		IF bFullPackage THEN
		//WXT530
			//Add collection WXT530
			IF GVL_Fastighet.WXT530 THEN
				M_AddJSONObject('CollectionOpen', 'WXT530');
				//Vind (aR1)
					M_AddJSONObject('DN', TO_STRING(GVL_WXT530._GW3U_DN));
					M_AddJSONObject('DM', TO_STRING(GVL_WXT530._GW3U_DM));
					M_AddJSONObject('DX', TO_STRING(GVL_WXT530._GW3U_DX));
					M_AddJSONObject('SN', TO_STRING(GVL_WXT530._GW3U_SN));
					M_AddJSONObject('SM', TO_STRING(GVL_WXT530._GW3U_SM));
					M_AddJSONObject('SX', TO_STRING(GVL_WXT530._GW3U_SX));
				//Tryck, temperatur och fuktighet (aR2)
					M_AddJSONObject('GT3U', TO_STRING(GVL_WXT530._GW3U_GT3U));
					M_AddJSONObject('GT41', TO_STRING(GVL_WXT530._GW3U_GT41));
					M_AddJSONObject('GM41', TO_STRING(GVL_WXT530._GW3U_GM41));
					M_AddJSONObject('GP41', TO_STRING(GVL_WXT530._GW3U_GP41));	
				//Nederbörd (aR3)		
					M_AddJSONObject('RC', TO_STRING(GVL_WXT530._GW3U_RC));
					M_AddJSONObject('RD', TO_STRING(GVL_WXT530._GW3U_RD));
					M_AddJSONObject('RI', TO_STRING(GVL_WXT530._GW3U_RI));
					M_AddJSONObject('HC', TO_STRING(GVL_WXT530._GW3U_HC));
					M_AddJSONObject('HD', TO_STRING(GVL_WXT530._GW3U_HD));
					M_AddJSONObject('HI', TO_STRING(GVL_WXT530._GW3U_HI));
					M_AddJSONObject('RP', TO_STRING(GVL_WXT530._GW3U_RP));
					M_AddJSONObject('HP', TO_STRING(GVL_WXT530._GW3U_HP));		
			//Close collection WXT530
				M_AddJSONObject('CollectionClose',',');
			END_IF
		//IO
			//Add collection IO
				M_AddJSONObject('CollectionOpen', 'IO');
				// Analog in, hårdvara
					//M_AddJSONObject('AI1', TO_STRING(GVL_IO._AI1));
					//M_AddJSONObject('AI2', TO_STRING(GVL_IO._AI2));
					//M_AddJSONObject('AI3', TO_STRING(GVL_IO._AI3));
					//M_AddJSONObject('AI4', TO_STRING(GVL_IO._AI4));
					//M_AddJSONObject('AI5', TO_STRING(GVL_IO._AI5));
					//M_AddJSONObject('AI6', TO_STRING(GVL_IO._AI6));
					//M_AddJSONObject('AI7', TO_STRING(GVL_IO._AI7));
					//M_AddJSONObject('AI8', TO_STRING(GVL_IO._AI8));
				// Analog in
					M_AddJSONObject('GT41_MV', TO_STRING(GVL_IO._GT41_MV / 100)); //Scaled to degrees celsius, PT1000 temp sensor at F15
					M_AddJSONObject('GT42_MV', TO_STRING(GVL_IO._GT42_MV / 100)); //Scaled to degrees celsius, PT1000 temp sensor at F15
					M_AddJSONObject('GT43_MV', TO_STRING(GVL_IO._GT43_MV));
					M_AddJSONObject('GT44_MV', TO_STRING(GVL_IO._GT44_MV));
					M_AddJSONObject('GT45_MV', TO_STRING(GVL_IO._GT45_MV));
					M_AddJSONObject('GT46_MV', TO_STRING(GVL_IO._GT46_MV));
					M_AddJSONObject('GT47_MV', TO_STRING(GVL_IO._GT47_MV));
					M_AddJSONObject('GT48_MV', TO_STRING(GVL_IO._GT48_MV));
			//Close collection IO
				M_AddJSONObject('CollectionClose',',');				
		END_IF
		//ClusterControl
			//Add new collection ClusterControl
				M_AddJSONObject('CollectionOpen', 'ClusterControl');		
				//V1
					//M_AddJSONObject('V1_IT', TO_STRING(GVL_ClusterCtrl._CCtrl_V1_IT));
					M_AddJSONObject('V1_P', TO_STRING(GVL_ClusterCtrl._CCtrl_V1_P));
					M_AddJSONObject('V1_P1', TO_STRING(GVL_ClusterCtrl._CCtrl_V1_P1));
					M_AddJSONObject('V1_P2', TO_STRING(GVL_ClusterCtrl._CCtrl_V1_P2));
					M_AddJSONObject('V1_P3', TO_STRING(GVL_ClusterCtrl._CCtrl_V1_P3));
					M_AddJSONObject('V1_U1_L1_N', TO_STRING(GVL_ClusterCtrl._CCtrl_V1_U1_L1_N));
					M_AddJSONObject('V1_U2_L2_N', TO_STRING(GVL_ClusterCtrl._CCtrl_V1_U2_L2_N));
					M_AddJSONObject('V1_U3_L3_N', TO_STRING(GVL_ClusterCtrl._CCtrl_V1_U3_L3_N));
					M_AddJSONObject('V1_U1_L1_L2', TO_STRING(GVL_ClusterCtrl._CCtrl_V1_U1_L1_L2));
					M_AddJSONObject('V1_U2_L2_L3', TO_STRING(GVL_ClusterCtrl._CCtrl_V1_U2_L2_L3));
					M_AddJSONObject('V1_U3_L3_L1', TO_STRING(GVL_ClusterCtrl._CCtrl_V1_U3_L3_L1));
					M_AddJSONObject('V1_Itot', TO_STRING(GVL_ClusterCtrl._CCtrl_V1_Itot));
					M_AddJSONObject('V1_I1', TO_STRING(GVL_ClusterCtrl._CCtrl_V1_I1));
					M_AddJSONObject('V1_I2', TO_STRING(GVL_ClusterCtrl._CCtrl_V1_I2));
					M_AddJSONObject('V1_I3', TO_STRING(GVL_ClusterCtrl._CCtrl_V1_I3));
					//M_AddJSONObject('V1_Yield_Wh', TO_STRING(GVL_ClusterCtrl._CCtrl_V1_Yield_Wh));
					M_AddJSONObject('V1_Yield_kWh', TO_STRING(GVL_ClusterCtrl._CCtrl_V1_Yield_kWh));
					M_AddJSONObject('V1_Yield_MWh', TO_STRING(GVL_ClusterCtrl._CCtrl_V1_Yield_MWh));
					//M_AddJSONObject('V1_YieldDay_Wh', TO_STRING(GVL_ClusterCtrl._CCtrl_V1_YieldDay_Wh));
					M_AddJSONObject('V1_YieldDay_kWh', TO_STRING(GVL_ClusterCtrl._CCtrl_V1_YieldDay_kWh));
					M_AddJSONObject('V1_PV', TO_STRING(GVL_ClusterCtrl._CCtrl_V1_PV));	
					M_AddJSONObject('V1_HZ', TO_STRING(GVL_ClusterCtrl._CCtrl_V1_HZ));			
				//V2
					//M_AddJSONObject('V2_IT', TO_STRING(GVL_ClusterCtrl._CCtrl_V2_IT));
					M_AddJSONObject('V2_P', TO_STRING(GVL_ClusterCtrl._CCtrl_V2_P));
					M_AddJSONObject('V2_P1', TO_STRING(GVL_ClusterCtrl._CCtrl_V2_P1));
					M_AddJSONObject('V2_P2', TO_STRING(GVL_ClusterCtrl._CCtrl_V2_P2));
					M_AddJSONObject('V2_P3', TO_STRING(GVL_ClusterCtrl._CCtrl_V2_P3));
					M_AddJSONObject('V2_U1_L1_N', TO_STRING(GVL_ClusterCtrl._CCtrl_V2_U1_L1_N));
					M_AddJSONObject('V2_U2_L2_N', TO_STRING(GVL_ClusterCtrl._CCtrl_V2_U2_L2_N));
					M_AddJSONObject('V2_U3_L3_N', TO_STRING(GVL_ClusterCtrl._CCtrl_V2_U3_L3_N));
					M_AddJSONObject('V2_U1_L1_L2', TO_STRING(GVL_ClusterCtrl._CCtrl_V2_U1_L1_L2));
					M_AddJSONObject('V2_U2_L2_L3', TO_STRING(GVL_ClusterCtrl._CCtrl_V2_U2_L2_L3));
					M_AddJSONObject('V2_U3_L3_L1', TO_STRING(GVL_ClusterCtrl._CCtrl_V2_U3_L3_L1));
					M_AddJSONObject('V2_Itot', TO_STRING(GVL_ClusterCtrl._CCtrl_V2_Itot));
					M_AddJSONObject('V2_I1', TO_STRING(GVL_ClusterCtrl._CCtrl_V2_I1));
					M_AddJSONObject('V2_I2', TO_STRING(GVL_ClusterCtrl._CCtrl_V2_I2));
					M_AddJSONObject('V2_I3', TO_STRING(GVL_ClusterCtrl._CCtrl_V2_I3));
					//M_AddJSONObject('V2_Yield_Wh', TO_STRING(GVL_ClusterCtrl._CCtrl_V2_Yield_Wh));
					M_AddJSONObject('V2_Yield_kWh', TO_STRING(GVL_ClusterCtrl._CCtrl_V2_Yield_kWh));
					M_AddJSONObject('V2_Yield_MWh', TO_STRING(GVL_ClusterCtrl._CCtrl_V2_Yield_MWh));
					//M_AddJSONObject('V2_YieldDay_Wh', TO_STRING(GVL_ClusterCtrl._CCtrl_V2_YieldDay_Wh));
					M_AddJSONObject('V2_YieldDay_kWh', TO_STRING(GVL_ClusterCtrl._CCtrl_V2_YieldDay_kWh));
					M_AddJSONObject('V2_PV', TO_STRING(GVL_ClusterCtrl._CCtrl_V2_PV));	
					M_AddJSONObject('V2_HZ', TO_STRING(GVL_ClusterCtrl._CCtrl_V2_HZ));	
				//V3
					//M_AddJSONObject('V3_IT', TO_STRING(GVL_ClusterCtrl._CCtrl_V3_IT));
					M_AddJSONObject('V3_P', TO_STRING(GVL_ClusterCtrl._CCtrl_V3_P));
					M_AddJSONObject('V3_P1', TO_STRING(GVL_ClusterCtrl._CCtrl_V3_P1));
					M_AddJSONObject('V3_P2', TO_STRING(GVL_ClusterCtrl._CCtrl_V3_P2));
					M_AddJSONObject('V3_P3', TO_STRING(GVL_ClusterCtrl._CCtrl_V3_P3));
					M_AddJSONObject('V3_U1_L1_N', TO_STRING(GVL_ClusterCtrl._CCtrl_V3_U1_L1_N));
					M_AddJSONObject('V3_U2_L2_N', TO_STRING(GVL_ClusterCtrl._CCtrl_V3_U2_L2_N));
					M_AddJSONObject('V3_U3_L3_N', TO_STRING(GVL_ClusterCtrl._CCtrl_V3_U3_L3_N));
					M_AddJSONObject('V3_U1_L1_L2', TO_STRING(GVL_ClusterCtrl._CCtrl_V3_U1_L1_L2));
					M_AddJSONObject('V3_U2_L2_L3', TO_STRING(GVL_ClusterCtrl._CCtrl_V3_U2_L2_L3));
					M_AddJSONObject('V3_U3_L3_L1', TO_STRING(GVL_ClusterCtrl._CCtrl_V3_U3_L3_L1));
					M_AddJSONObject('V3_Itot', TO_STRING(GVL_ClusterCtrl._CCtrl_V3_Itot));
					M_AddJSONObject('V3_I1', TO_STRING(GVL_ClusterCtrl._CCtrl_V3_I1));
					M_AddJSONObject('V3_I2', TO_STRING(GVL_ClusterCtrl._CCtrl_V3_I2));
					M_AddJSONObject('V3_I3', TO_STRING(GVL_ClusterCtrl._CCtrl_V3_I3));
					//M_AddJSONObject('V3_Yield_Wh', TO_STRING(GVL_ClusterCtrl._CCtrl_V3_Yield_Wh));
					M_AddJSONObject('V3_Yield_kWh', TO_STRING(GVL_ClusterCtrl._CCtrl_V3_Yield_kWh));
					M_AddJSONObject('V3_Yield_MWh', TO_STRING(GVL_ClusterCtrl._CCtrl_V3_Yield_MWh));
					//M_AddJSONObject('V3_YieldDay_Wh', TO_STRING(GVL_ClusterCtrl._CCtrl_V3_YieldDay_Wh));
					M_AddJSONObject('V3_YieldDay_kWh', TO_STRING(GVL_ClusterCtrl._CCtrl_V3_YieldDay_kWh));
					M_AddJSONObject('V3_PV', TO_STRING(GVL_ClusterCtrl._CCtrl_V3_PV));	
					M_AddJSONObject('V3_HZ', TO_STRING(GVL_ClusterCtrl._CCtrl_V3_HZ));	
			//Close collection ClusterControl
				M_AddJSONObject('CollectionClose',',');	
		//MX41
			//Add new collection MX41
				M_AddJSONObject('CollectionOpen', 'MX41');
				//MX41 Data
					M_AddJSONObject('I1', TO_STRING(GVL_MX41._I1));
					M_AddJSONObject('I2', TO_STRING(GVL_MX41._I2));
					M_AddJSONObject('I3', TO_STRING(GVL_MX41._I3));
					M_AddJSONObject('U1_U2', TO_STRING(GVL_MX41._U1_U2));
					M_AddJSONObject('U2_U3', TO_STRING(GVL_MX41._U2_U3));
					M_AddJSONObject('U3_U1', TO_STRING(GVL_MX41._U3_U1));
					M_AddJSONObject('U1_N', TO_STRING(GVL_MX41._U1_N));
					M_AddJSONObject('U2_N', TO_STRING(GVL_MX41._U2_N));
					M_AddJSONObject('U3_N', TO_STRING(GVL_MX41._U3_N));
					M_AddJSONObject('P1', TO_STRING(GVL_MX41._P1));
					M_AddJSONObject('P2', TO_STRING(GVL_MX41._P2));
					M_AddJSONObject('P3', TO_STRING(GVL_MX41._P3));
					M_AddJSONObject('P', TO_STRING(GVL_MX41._P));
					M_AddJSONObject('PVAR', TO_STRING(GVL_MX41._PVAR));
					M_AddJSONObject('PVA', TO_STRING(GVL_MX41._PVA));
					M_AddJSONObject('PFA', TO_STRING(GVL_MX41._Pfa));
					M_AddJSONObject('HZ', TO_STRING(GVL_MX41._HZ));
					M_AddJSONObject('WHAI', TO_STRING(GVL_MX41._WHAI));
					M_AddJSONObject('WHAE', TO_STRING(GVL_MX41._WHAE));
					M_AddJSONObject('VARHI', TO_STRING(GVL_MX41._VARHI));
					M_AddJSONObject('VARHE', TO_STRING(GVL_MX41._VARHE));
					M_AddJSONObject('WHPAI', TO_STRING(GVL_MX41._WHPAI));
					M_AddJSONObject('WHPAE', TO_STRING(GVL_MX41._WHPAE));
					M_AddJSONObject('WHAEI1', TO_STRING(GVL_MX41._WHAEI1));
					M_AddJSONObject('WHAEI2', TO_STRING(GVL_MX41._WHAEI2));
					M_AddJSONObject('WHAEI3', TO_STRING(GVL_MX41._WHAEI3));
			//Close collection MX41	
				M_AddJSONObject('CollectionClose',',');	
		//SR05 Hukseflux Solar Irradiance meter
		IF GVL_Fastighet.SMAIrrMeter THEN
			//Add collection SR05
				M_AddJSONObject('CollectionOpen', 'SR05');
				//SR05 Sensor Outputs
					M_AddJSONObject('Irr', TO_STRING(GVL_SR05._SolarIrr));
					M_AddJSONObject('BT', TO_STRING(GVL_SR05._BodyTemp));
					M_AddJSONObject('ER', TO_STRING(GVL_SR05._ElecResistance));
					M_AddJSONObject('VO', TO_STRING(GVL_SR05._VoltageOutput));					
			//Close collection SR05
				M_AddJSONObject('End', sCurlyBracketEnd);
		END_IF
	//Close collection DataList	
		M_AddJSONObject('End', sCurlyBracketEnd);	
	//////////////////////////////////////////
	
	//End Collection
	M_AddJSONObject('End', sCurlyBracketEnd);	

	//Done
	M_BuildPayload := TRUE;
END_METHOD

METHOD M_ConnectMQTT : BOOL
VAR_INPUT
END_VAR
bConnect := TRUE;
END_METHOD

METHOD M_CreatePayload : BOOL
VAR_INPUT
	bFullPackage : BOOL;
END_VAR
VAR
	nLastPosAdded : DINT;
	i : DINT;
	sStringCheck : STRING;
	M_Payload_SMAClusterCntrl: INT;
END_VAR
// Method for building the Payload message that is going to be sent to the Azure IoT Hub. 
// Maximum 4kB message 
		
//Clear Payload before creating a new one
uPayload := GVL_IoT.uPayloadEmpty;

//Start Collection
M_AddJSONObject('Start', sCurlyBracket);

//General
M_AddJSONObject('ID', GVL_Fastighet.FastighetsBeteckning);
M_AddJSONObject('timeStamp', sJSONTime);

//Add new collection DataList
M_AddJSONObject('CollectionOpen', 'DataList');

(* Add the units payload that are enabled *)
IF bFullPackage THEN
	
	IF GVL_Fastighet.WXT530 THEN
		M_Payload_WXT530();
	END_IF
	
	IF GVL_Fastighet.IO THEN
		M_Payload_IO();
	END_IF
	
END_IF

IF GVL_Fastighet.SMAClusterCntrl THEN
		M_Payload_SMACluster();
END_IF

IF GVL_Fastighet.EnergyMeter THEN
	M_Payload_MX41_iEM3255();
END_IF

IF GVL_Fastighet.SR05 THEN
	M_Payload_SR05();
END_IF

//Trim the payload char ',' from last unit added to create a valid json
//Check first empty position in the array
FOR i:=0 TO SIZEOF(uPayLoad.aPayload) / SIZEOF(uPayload.aPayload[0]) DO
	IF uPayload.aPayload[i] = 0 THEN
		nLastPosAdded := i;
		EXIT;
	END_IF
END_FOR

//Remove the last ',' char to make a valid json-string
uPayload.aPayload[nLastPosAdded - 1] := 0;


//Close collection DataList	
M_AddJSONObject('End', sCurlyBracketEnd);	

//End Collection
M_AddJSONObject('End', sCurlyBracketEnd);	

//Done
M_CreatePayload := TRUE;
END_METHOD

METHOD M_Deque : BOOL
VAR
	i : INT;
END_VAR
FOR i:=0 TO GVL_IoT.nMaxPayloadBuffer DO

	//If there is data, publish it! 
	IF MEMCMP(ADR(GVL_IoT.uPayloadQueue[i]), ADR(GVL_IoT.uPayloadEmpty), SIZEOF(GVL_IoT.uPayloadEmpty)) <> 0 THEN
		//Call Publish 
		M_Publish(GVL_IoT.uPayloadQueue[i]);
		//After the publish; remove it from the queue
		GVL_IoT.uPayloadQueue[i] := GVL_IoT.uPayloadEmpty;
	END_IF

END_FOR

//Done
M_Deque := TRUE;
END_METHOD

METHOD M_DisconnectMQTT : BOOL
VAR_INPUT
END_VAR
bConnect := FALSE;
END_METHOD

METHOD M_Initialize : BOOL
VAR_INPUT
END_VAR
//Initialize startup parameters

	//Message topic that is used for every message, should not be changed! Only if the deviceName have changed
	sTopicPub := GVL_Fastighet.IoTTopicPub;
	
	//Set the SAS token
	fbMqttClient.sHostName := GVL_Fastighet.IoTHostName;
	fbMqttClient.nHostPort := GVL_Fastighet.IoTHostPort;
	//fbMqttClient.stTLS.sAzureSas := 'HostName=StunsSolarHub.azure-devices.net;DeviceId=SE_UPP_A001P001;SharedAccessSignature=SharedAccessSignature sr=StunsSolarHub.azure-devices.net%2Fdevices%2FSE_UPP_A001P001&sig=PNxS244bUszDXJ%2BMNceHTcws%2BEW3ixqGkw0V7mblAEw%3D&se=1525956832';
	//fbMqttClient.stTLS.sCA := 'c:\TwinCAT\3.1\Config\Certificates\azure.crt';
	
	//Default Publish time
	tPublishTime(PT:=GVL_Fastighet.PublishTime);

	//Set Active flag
	bActive:= TRUE;

//Initialize completed
	bInitDone := TRUE;
END_METHOD

METHOD M_Payload_IO : BOOL
VAR_INPUT
END_VAR
//IO
//Add collection IO
M_AddJSONObject('CollectionOpen', 'IO');
// Analog in
M_AddJSONObject('GT41_MV', TO_STRING(GVL_IO._GT41_MV / 100)); //Scaled to degrees celsius, PT1000 temp sensor at F15
M_AddJSONObject('GT42_MV', TO_STRING(GVL_IO._GT42_MV / 100)); //Scaled to degrees celsius, PT1000 temp sensor at F15
M_AddJSONObject('GT43_MV', TO_STRING(GVL_IO._GT43_MV));
M_AddJSONObject('GT44_MV', TO_STRING(GVL_IO._GT44_MV));
M_AddJSONObject('GT45_MV', TO_STRING(GVL_IO._GT45_MV));
M_AddJSONObject('GT46_MV', TO_STRING(GVL_IO._GT46_MV));
M_AddJSONObject('GT47_MV', TO_STRING(GVL_IO._GT47_MV));
M_AddJSONObject('GT48_MV', TO_STRING(GVL_IO._GT48_MV));
//Close collection IO
M_AddJSONObject('CollectionClose',',');
END_METHOD

METHOD M_Payload_MX41_iEM3255 : BOOL
VAR_INPUT
END_VAR
//Add collection MX41
M_AddJSONObject('CollectionOpen', 'MX41');

//MX41 Data - Schneider
M_AddJSONObject('I1', TO_STRING(GVL_MX41._I1));
M_AddJSONObject('I2', TO_STRING(GVL_MX41._I2));
M_AddJSONObject('I3', TO_STRING(GVL_MX41._I3));
M_AddJSONObject('U1_U2', TO_STRING(GVL_MX41._U1_U2));
M_AddJSONObject('U2_U3', TO_STRING(GVL_MX41._U2_U3));
M_AddJSONObject('U3_U1', TO_STRING(GVL_MX41._U3_U1));
(*The following voltage values only returns 0 at F15 per 20017-09-01, investigate and remove commentation when working. Possibly lack of N leader to meter!*)
//M_AddJSONObject('U1_N', TO_STRING(GVL_MX41._U1_N));
//M_AddJSONObject('U2_N', TO_STRING(GVL_MX41._U2_N));
//M_AddJSONObject('U3_N', TO_STRING(GVL_MX41._U3_N));
(*The following power values only returns 0 at F15 per 20017-09-01, investigate and remove commentation when working. Possibly lack of N leader to meter!*)
//M_AddJSONObject('P1', TO_STRING(GVL_MX41._P1));
//M_AddJSONObject('P2', TO_STRING(GVL_MX41._P2));
//M_AddJSONObject('P3', TO_STRING(GVL_MX41._P3));
M_AddJSONObject('P', TO_STRING(GVL_MX41._P));
M_AddJSONObject('PVAR', TO_STRING(GVL_MX41._PVAR));
M_AddJSONObject('PVA', TO_STRING(GVL_MX41._PVA));
M_AddJSONObject('PFA', TO_STRING(GVL_MX41._Pfa));
M_AddJSONObject('HZ', TO_STRING(GVL_MX41._HZ));
M_AddJSONObject('WHAI', TO_STRING(GVL_MX41._WHAI));
M_AddJSONObject('WHAE', TO_STRING(GVL_MX41._WHAE));
M_AddJSONObject('VARHI', TO_STRING(GVL_MX41._VARHI));
M_AddJSONObject('VARHE', TO_STRING(GVL_MX41._VARHE));
M_AddJSONObject('WHPAI', TO_STRING(GVL_MX41._WHPAI));
M_AddJSONObject('WHPAE', TO_STRING(GVL_MX41._WHPAE));
M_AddJSONObject('WHAEI1', TO_STRING(GVL_MX41._WHAEI1));
M_AddJSONObject('WHAEI2', TO_STRING(GVL_MX41._WHAEI2));
M_AddJSONObject('WHAEI3', TO_STRING(GVL_MX41._WHAEI3));

//Close collection MX41	
M_AddJSONObject('CollectionClose',',');
END_METHOD

METHOD M_Payload_SMACluster : BOOL
VAR_INPUT
END_VAR
//Add new collection ClusterControl
M_AddJSONObject('CollectionOpen', 'ClusterControl');		


//V1 - Inverter 1
//M_AddJSONObject('V1_IT', TO_STRING(GVL_ClusterCtrl._CCtrl_V1_IT));
M_AddJSONObject('V1_P', TO_STRING(GVL_ClusterCtrl._CCtrl_V1_P));
M_AddJSONObject('V1_P1', TO_STRING(GVL_ClusterCtrl._CCtrl_V1_P1));
M_AddJSONObject('V1_P2', TO_STRING(GVL_ClusterCtrl._CCtrl_V1_P2));
M_AddJSONObject('V1_P3', TO_STRING(GVL_ClusterCtrl._CCtrl_V1_P3));
M_AddJSONObject('V1_U1_L1_N', TO_STRING(GVL_ClusterCtrl._CCtrl_V1_U1_L1_N));
M_AddJSONObject('V1_U2_L2_N', TO_STRING(GVL_ClusterCtrl._CCtrl_V1_U2_L2_N));
M_AddJSONObject('V1_U3_L3_N', TO_STRING(GVL_ClusterCtrl._CCtrl_V1_U3_L3_N));
(*The following voltage values only returns false values at F15 per 20017-09-01, investigate and remove commentation when working*)
//M_AddJSONObject('V1_U1_L1_L2', TO_STRING(GVL_ClusterCtrl._CCtrl_V1_U1_L1_L2));
//M_AddJSONObject('V1_U2_L2_L3', TO_STRING(GVL_ClusterCtrl._CCtrl_V1_U2_L2_L3));
//M_AddJSONObject('V1_U3_L3_L1', TO_STRING(GVL_ClusterCtrl._CCtrl_V1_U3_L3_L1));
(*The following parameter Itot only returns a false value at F15 per 20017-09-01, investigate and remove commentation when working*)
//M_AddJSONObject('V1_Itot', TO_STRING(GVL_ClusterCtrl._CCtrl_V1_Itot));
M_AddJSONObject('V1_I1', TO_STRING(GVL_ClusterCtrl._CCtrl_V1_I1));
M_AddJSONObject('V1_I2', TO_STRING(GVL_ClusterCtrl._CCtrl_V1_I2));
M_AddJSONObject('V1_I3', TO_STRING(GVL_ClusterCtrl._CCtrl_V1_I3));
//M_AddJSONObject('V1_Yield_Wh', TO_STRING(GVL_ClusterCtrl._CCtrl_V1_Yield_Wh));
M_AddJSONObject('V1_Yield_kWh', TO_STRING(GVL_ClusterCtrl._CCtrl_V1_Yield_kWh));
M_AddJSONObject('V1_Yield_MWh', TO_STRING(GVL_ClusterCtrl._CCtrl_V1_Yield_MWh));
//M_AddJSONObject('V1_YieldDay_Wh', TO_STRING(GVL_ClusterCtrl._CCtrl_V1_YieldDay_Wh));
M_AddJSONObject('V1_YieldDay_kWh', TO_STRING(GVL_ClusterCtrl._CCtrl_V1_YieldDay_kWh));
(*The following parameter PV only returns a false value at F15 per 20017-09-01, investigate and remove commentation when working*)
//M_AddJSONObject('V1_PV', TO_STRING(GVL_ClusterCtrl._CCtrl_V1_PV));	
M_AddJSONObject('V1_HZ', TO_STRING(GVL_ClusterCtrl._CCtrl_V1_HZ));			


//V2 - Inverter 2
//M_AddJSONObject('V2_IT', TO_STRING(GVL_ClusterCtrl._CCtrl_V2_IT));
M_AddJSONObject('V2_P', TO_STRING(GVL_ClusterCtrl._CCtrl_V2_P));
M_AddJSONObject('V2_P1', TO_STRING(GVL_ClusterCtrl._CCtrl_V2_P1));
M_AddJSONObject('V2_P2', TO_STRING(GVL_ClusterCtrl._CCtrl_V2_P2));
M_AddJSONObject('V2_P3', TO_STRING(GVL_ClusterCtrl._CCtrl_V2_P3));
M_AddJSONObject('V2_U1_L1_N', TO_STRING(GVL_ClusterCtrl._CCtrl_V2_U1_L1_N));
M_AddJSONObject('V2_U2_L2_N', TO_STRING(GVL_ClusterCtrl._CCtrl_V2_U2_L2_N));
M_AddJSONObject('V2_U3_L3_N', TO_STRING(GVL_ClusterCtrl._CCtrl_V2_U3_L3_N));
(*The following voltage values only return false values at F15 per 20017-09-01, investigate and remove commentation when working*)
//M_AddJSONObject('V2_U1_L1_L2', TO_STRING(GVL_ClusterCtrl._CCtrl_V2_U1_L1_L2));
//M_AddJSONObject('V2_U2_L2_L3', TO_STRING(GVL_ClusterCtrl._CCtrl_V2_U2_L2_L3));
//M_AddJSONObject('V2_U3_L3_L1', TO_STRING(GVL_ClusterCtrl._CCtrl_V2_U3_L3_L1));
(*The following parameter Itot only returns a false value at F15 per 20017-09-01, investigate and remove commentation when working*)
//M_AddJSONObject('V2_Itot', TO_STRING(GVL_ClusterCtrl._CCtrl_V2_Itot));
M_AddJSONObject('V2_I1', TO_STRING(GVL_ClusterCtrl._CCtrl_V2_I1));
M_AddJSONObject('V2_I2', TO_STRING(GVL_ClusterCtrl._CCtrl_V2_I2));
M_AddJSONObject('V2_I3', TO_STRING(GVL_ClusterCtrl._CCtrl_V2_I3));
//M_AddJSONObject('V2_Yield_Wh', TO_STRING(GVL_ClusterCtrl._CCtrl_V2_Yield_Wh));
M_AddJSONObject('V2_Yield_kWh', TO_STRING(GVL_ClusterCtrl._CCtrl_V2_Yield_kWh));
M_AddJSONObject('V2_Yield_MWh', TO_STRING(GVL_ClusterCtrl._CCtrl_V2_Yield_MWh));
//M_AddJSONObject('V2_YieldDay_Wh', TO_STRING(GVL_ClusterCtrl._CCtrl_V2_YieldDay_Wh));
M_AddJSONObject('V2_YieldDay_kWh', TO_STRING(GVL_ClusterCtrl._CCtrl_V2_YieldDay_kWh));
(*The following parameter PV only returns a false value at F15 per 20017-09-01, investigate and remove commentation when working*)
//M_AddJSONObject('V2_PV', TO_STRING(GVL_ClusterCtrl._CCtrl_V2_PV));	
M_AddJSONObject('V2_HZ', TO_STRING(GVL_ClusterCtrl._CCtrl_V2_HZ));	

//V3 - Inverter 3
//M_AddJSONObject('V3_IT', TO_STRING(GVL_ClusterCtrl._CCtrl_V3_IT));
M_AddJSONObject('V3_P', TO_STRING(GVL_ClusterCtrl._CCtrl_V3_P));
M_AddJSONObject('V3_P1', TO_STRING(GVL_ClusterCtrl._CCtrl_V3_P1));
M_AddJSONObject('V3_P2', TO_STRING(GVL_ClusterCtrl._CCtrl_V3_P2));
M_AddJSONObject('V3_P3', TO_STRING(GVL_ClusterCtrl._CCtrl_V3_P3));
M_AddJSONObject('V3_U1_L1_N', TO_STRING(GVL_ClusterCtrl._CCtrl_V3_U1_L1_N));
M_AddJSONObject('V3_U2_L2_N', TO_STRING(GVL_ClusterCtrl._CCtrl_V3_U2_L2_N));
M_AddJSONObject('V3_U3_L3_N', TO_STRING(GVL_ClusterCtrl._CCtrl_V3_U3_L3_N));
(*The following voltage values only return false values at F15 per 20017-09-01, investigate and remove commentation when working*)
//M_AddJSONObject('V3_U1_L1_L2', TO_STRING(GVL_ClusterCtrl._CCtrl_V3_U1_L1_L2));
//M_AddJSONObject('V3_U2_L2_L3', TO_STRING(GVL_ClusterCtrl._CCtrl_V3_U2_L2_L3));
//M_AddJSONObject('V3_U3_L3_L1', TO_STRING(GVL_ClusterCtrl._CCtrl_V3_U3_L3_L1));
(*The following parameter Itot only returns a false value at F15 per 20017-09-01, investigate and remove commentation when working*)
//M_AddJSONObject('V3_Itot', TO_STRING(GVL_ClusterCtrl._CCtrl_V3_Itot));
M_AddJSONObject('V3_I1', TO_STRING(GVL_ClusterCtrl._CCtrl_V3_I1));
M_AddJSONObject('V3_I2', TO_STRING(GVL_ClusterCtrl._CCtrl_V3_I2));
M_AddJSONObject('V3_I3', TO_STRING(GVL_ClusterCtrl._CCtrl_V3_I3));
//M_AddJSONObject('V3_Yield_Wh', TO_STRING(GVL_ClusterCtrl._CCtrl_V3_Yield_Wh));
M_AddJSONObject('V3_Yield_kWh', TO_STRING(GVL_ClusterCtrl._CCtrl_V3_Yield_kWh));
M_AddJSONObject('V3_Yield_MWh', TO_STRING(GVL_ClusterCtrl._CCtrl_V3_Yield_MWh));
//M_AddJSONObject('V3_YieldDay_Wh', TO_STRING(GVL_ClusterCtrl._CCtrl_V3_YieldDay_Wh));
M_AddJSONObject('V3_YieldDay_kWh', TO_STRING(GVL_ClusterCtrl._CCtrl_V3_YieldDay_kWh));
(*The following parameter PV only returns a false value at F15 per 20017-09-01, investigate and remove commentation when working*)
//M_AddJSONObject('V3_PV', TO_STRING(GVL_ClusterCtrl._CCtrl_V3_PV));	
M_AddJSONObject('V3_HZ', TO_STRING(GVL_ClusterCtrl._CCtrl_V3_HZ));	


//Close collection ClusterControl
M_AddJSONObject('CollectionClose',',');
END_METHOD

METHOD M_Payload_SMAIrrMeter : BOOL
VAR_INPUT
END_VAR
END_METHOD

METHOD M_Payload_SR05 : BOOL
VAR_INPUT
END_VAR
//SR05 Hukseflux Solar Irradiance meter
//Add collection SR05
M_AddJSONObject('CollectionOpen', 'SR05');
//SR05 Sensor Outputs
M_AddJSONObject('Irr', TO_STRING(GVL_SR05._SolarIrr));
M_AddJSONObject('TempBody', TO_STRING(GVL_SR05._BodyTemp));
M_AddJSONObject('ElectricalRes', TO_STRING(GVL_SR05._ElecResistance));
M_AddJSONObject('VoltageOutput', TO_STRING(GVL_SR05._VoltageOutput));					
//Close collection SR05
M_AddJSONObject('CollectionClose',',');
END_METHOD

METHOD M_Payload_WXT530 : BOOL
VAR_INPUT
END_VAR
//WXT530
//Add collection WXT530
M_AddJSONObject('CollectionOpen', 'WXT530');
//Vind (aR1)
M_AddJSONObject('DN', TO_STRING(GVL_WXT530._GW3U_DN));
M_AddJSONObject('DM', TO_STRING(GVL_WXT530._GW3U_DM));
M_AddJSONObject('DX', TO_STRING(GVL_WXT530._GW3U_DX));
M_AddJSONObject('SN', TO_STRING(GVL_WXT530._GW3U_SN));
M_AddJSONObject('SM', TO_STRING(GVL_WXT530._GW3U_SM));
M_AddJSONObject('SX', TO_STRING(GVL_WXT530._GW3U_SX));
//Tryck, temperatur och fuktighet (aR2)
M_AddJSONObject('GT3U', TO_STRING(GVL_WXT530._GW3U_GT3U));
M_AddJSONObject('GT41', TO_STRING(GVL_WXT530._GW3U_GT41));
M_AddJSONObject('GM41', TO_STRING(GVL_WXT530._GW3U_GM41));
M_AddJSONObject('GP41', TO_STRING(GVL_WXT530._GW3U_GP41));	
//Nederbörd (aR3)		
M_AddJSONObject('RC', TO_STRING(GVL_WXT530._GW3U_RC));
M_AddJSONObject('RD', TO_STRING(GVL_WXT530._GW3U_RD));
M_AddJSONObject('RI', TO_STRING(GVL_WXT530._GW3U_RI));
M_AddJSONObject('HC', TO_STRING(GVL_WXT530._GW3U_HC));
M_AddJSONObject('HD', TO_STRING(GVL_WXT530._GW3U_HD));
M_AddJSONObject('HI', TO_STRING(GVL_WXT530._GW3U_HI));
M_AddJSONObject('RP', TO_STRING(GVL_WXT530._GW3U_RP));
M_AddJSONObject('HP', TO_STRING(GVL_WXT530._GW3U_HP));		
//Close collection WXT530
M_AddJSONObject('CollectionClose',',');
END_METHOD

METHOD M_Publish : BOOL
VAR_INPUT
	uPayloadToPublish : U_Payload;
END_VAR
//Publish the payload
fbMqttClient.Publish(sTopic:= sTopicPub, 
									pPayload:= ADR(uPayloadToPublish.aPayload), 
									nPayloadSize:= SIZEOF(uPayloadToPublish.aPayload), 
									eQoS:= TcIotMqttQos.AtMostOnceDelivery, 
									bRetain:= FALSE, 
									bQueue:= FALSE );
//Update last published time
sLastPublishedTime := sSystemTime;		
//Increase the Publish counter
GVL_IoT.nTotalMessagePublished := GVL_IoT.nTotalMessagePublished + 1;
//Done								
M_Publish := TRUE;
END_METHOD

METHOD M_Queue : BOOL
VAR_INPUT
	uPayloadQueue : U_Payload;
END_VAR
//Check where to add it
IF GVL_IoT.nLastPos < GVL_IoT.nMaxPayloadBuffer THEN
	GVL_IoT.uPayloadQueue[GVL_IoT.nLastPos] := uPayloadQueue; //Add to buffer
END_IF

IF (GVL_IoT.nLastPos + 1) = GVL_IoT.nMaxPayloadBuffer THEN
	GVL_IoT.bBufferFull := TRUE;
ELSE
	GVL_IoT.bBufferFull := FALSE;
END_IF

//Done
M_Queue := TRUE;
END_METHOD

METHOD M_QueueBufferStatus
VAR
	i : INT;
END_VAR
//Check first empty position in the array
FOR i:=0 TO GVL_IoT.nMaxPayloadBuffer DO
	IF MEMCMP(ADR(GVL_IoT.uPayloadQueue[i]), ADR(GVL_IoT.uPayloadEmpty), SIZEOF(GVL_IoT.uPayloadEmpty)) = 1 THEN
		GVL_IoT.nLastPos := i;
		EXIT;
	END_IF
END_FOR

IF MEMCMP(ADR(GVL_IoT.uPayloadQueue[0]), ADR(GVL_IoT.uPayloadEmpty), SIZEOF(GVL_IoT.uPayloadEmpty)) = 1 THEN
	GVL_IoT.bBufferEmpty := TRUE;
ELSE
	GVL_IoT.bBufferEmpty := FALSE;
END_IF
END_METHOD

END_FUNCTION_BLOCK

// ---- POUs/Loggning/iEM3255_Logg.TcPOU
PROGRAM iEM3255_Logg
VAR
	
	fbLogg1 		:FB_SaveToCSV_Schneider;
	tUpdateTime1	:TIME:=T#5S;
	sFileName1		:STRING(255):='Schneider1';
	
	fbLogg2 		:FB_SaveToCSV_Schneider;
	tUpdateTime2	:TIME:=T#5S;
	sFileName2		:STRING(255):='Schneider2';
	
	fbLogg3 		:FB_SaveToCSV_Schneider;
	tUpdateTime3	:TIME:=T#5S;
	sFileName3		:STRING(255):='Schneider3';
	
	fbLogg4 		:FB_SaveToCSV_Schneider;
	tUpdateTime4	:TIME:=T#5S;
	sFileName4		:STRING(255):='Schneider4';

	
END_VAR

fbLogg1(
	bChangeSeparatorToComma:= FALSE, 
	bExecute:= GVL_Fastighet.CSVEnergyMeter, 
	tUpdateTime:= tUpdateTime1, 
	sFileName:= sFileName1, 
	nDayOfWeek:= PLC_TID.fbTime.systemTime.wDayOfWeek,
	sColumn1TimeStamp:= PLC_TID.systemTime, 
	sColumn2:= REAL_TO_STRING(GVL_MX41._I1), 
	sColumn3:= REAL_TO_STRING(GVL_MX41._I2), 
	sColumn4:= REAL_TO_STRING(GVL_MX41._I3), 
	sColumn5:= REAL_TO_STRING(GVL_MX41._U1_U2), 
	sColumn6:= REAL_TO_STRING(GVL_MX41._U2_U3), 
	sColumn7:= REAL_TO_STRING(GVL_MX41._U3_U1));
	
fbLogg2(
	bChangeSeparatorToComma:= FALSE, 
	bExecute:= GVL_Fastighet.CSVEnergyMeter, 
	tUpdateTime:= tUpdateTime2, 
	sFileName:= sFileName2, 
	nDayOfWeek:= PLC_TID.fbTime.systemTime.wDayOfWeek,
	sColumn1TimeStamp:= PLC_TID.systemTime, 
	sColumn2:= REAL_TO_STRING(GVL_MX41._P1), 
	sColumn3:= REAL_TO_STRING(GVL_MX41._P2), 
	sColumn4:= REAL_TO_STRING(GVL_MX41._P3), 
	sColumn5:= REAL_TO_STRING(GVL_MX41._PVAR), 
	sColumn6:= REAL_TO_STRING(GVL_MX41._PVA), 
	sColumn7:= REAL_TO_STRING(GVL_MX41._Pfa));
	
fbLogg3(
	bChangeSeparatorToComma:= FALSE, 
	bExecute:= GVL_Fastighet.CSVEnergyMeter, 
	tUpdateTime:= tUpdateTime3, 
	sFileName:= sFileName3, 
	nDayOfWeek:= PLC_TID.fbTime.systemTime.wDayOfWeek,
	sColumn1TimeStamp:= PLC_TID.systemTime, 
	sColumn2:= REAL_TO_STRING(GVL_MX41._HZ), 
	sColumn3:= REAL_TO_STRING(GVL_MX41._WHAI), 
	sColumn4:= REAL_TO_STRING(GVL_MX41._WHAE), 
	sColumn5:= REAL_TO_STRING(GVL_MX41._VARHI), 
	sColumn6:= REAL_TO_STRING(GVL_MX41._VARHE), 
	sColumn7:= REAL_TO_STRING(GVL_MX41._WHPAI));
	
fbLogg4(
	bChangeSeparatorToComma:= FALSE, 
	bExecute:= GVL_Fastighet.CSVEnergyMeter, 
	tUpdateTime:= tUpdateTime4, 
	sFileName:= sFileName4, 
	nDayOfWeek:= PLC_TID.fbTime.systemTime.wDayOfWeek,
	sColumn1TimeStamp:= PLC_TID.systemTime, 
	sColumn2:= REAL_TO_STRING(GVL_MX41._WHPAE), 
	sColumn3:= REAL_TO_STRING(GVL_MX41._WHAEI1), 
	sColumn4:= REAL_TO_STRING(GVL_MX41._WHAEI2), 
	sColumn5:= REAL_TO_STRING(GVL_MX41._WHAEI3),
	sColumn6:= REAL_TO_STRING(GVL_MX41._P));

END_PROGRAM

// ---- POUs/_FBs/FB_SaveToCSV_Schneider.TcPOU
FUNCTION_BLOCK FB_SaveToCSV_Schneider
VAR CONSTANT
	MAX_CSV_COLUMNS 	: UDINT := 7;
END_VAR
VAR_INPUT
	(*	In USA/UK the CSV field separator is a comma.
	In Germany and some other European countries the CSV field separator is a semicolon. *)
	bChangeSeparatorToComma	: BOOL := FALSE;
	bExecute : BOOL;
	tUpdateTime : TIME:=T#1S; //Update time 
	sFileName	: T_MaxString := 'DefaultName';(* CSV destination file path and name *)
	nDayOfWeek : WORD;
	sColumn1TimeStamp : T_MaxString;
	sColumn2 : STRING;
	sColumn3 : STRING;
	sColumn4 : STRING; 
	sColumn5 : STRING;
	sColumn6 : STRING;
	sColumn7 : STRING;
END_VAR
VAR
	sNetId			: T_AmsNetId := '';	(* TwinCAT system network address *)	
	sCSVLine		: T_MaxString := '';(* Single CSV text line (row, record), we are using string as record buffer (your are able to see created fields) *)
	sCSVField		: T_MaxString := '';(* Single CSV field value (column, record field) *)
	bBusy			: BOOL;
	bError			: BOOL;
	nErrId			: UDINT;
	nColumn		: UDINT 	:= 1;(* Column number (record field) *)
	hFile			: UINT		:= 0;(* File handle of the source file *)
	step			: DWORD 	:= 0;
	fbFileOpen	: FB_FileOpen;(* Opens file *)
	fbFileClose	: FB_FileClose;(* Closes file *)
	fbFilePuts		: FB_FilePuts;(* Writes one record (line) *)
	fbWriter		: FB_CSVMemBufferWriter;(* Helper function block used to create CSV data bytes (single record line) *)	
	tUpdateTimer : TON;
	sCompleteFileName : STRING;
	sPathName : T_MaxString;
	sTempDate : STRING;
	sDate : STRING;
	bWeekUpdate : BOOL;
END_VAR

(* Call the timer every plc-cycle *)
tUpdateTimer(IN:=NOT tUpdateTimer.Q, PT:=tUpdateTime);


(* Update filename *)
IF nDayOfWeek = 1 AND bWeekUpdate THEN //1=Monday	
		sCompleteFileName	:= sFileName;
		sTempDate := DELETE(sColumn1TimeStamp, 16,11); //Cut the timestamp so we only save the date
		sDate := INSERT(sTempDate, '_', 10); //Add '-' after the date for seperation
		sPathName:=CONCAT(CONCAT('C:\Loggning\Schneider\',CONCAT(sDate,sFileName)),'.csv');
		bWeekUpdate := FALSE;
ELSE
	(* Update if name has changed *)
	IF sCompleteFileName <> sFileName THEN
		sCompleteFileName := sFileName;
		sTempDate := DELETE(sColumn1TimeStamp, 16,11); //Cut the timestamp so we only save the date
		sDate := INSERT(sTempDate, '_', 10); //Add '-' after the date for seperation
		sPathName:=CONCAT(CONCAT('C:\Loggning\Schneider\',CONCAT(sDate,sCompleteFileName)),'.csv');
	END_IF	
END_IF

IF nDayOfWeek <> 1 THEN
	bWeekUpdate := TRUE;
END_IF

CASE step OF
	0:	(* Wait for rising edge at bWrite variable *)
		IF bExecute AND tUpdateTimer.Q THEN
			bBusy 		:= TRUE;
			bError		:= FALSE;
			nErrId		:= 0;
			hFile			:= 0;
			step 		:= 1;
		END_IF

	1:	(* Open source file *)
		fbFileOpen(  bExecute := FALSE  );
		fbFileOpen( 	sNetId := sNetId, sPathName := sPathName, nMode := FOPEN_MODEAPPEND OR FOPEN_MODETEXT,(* Open file in TEXT mode! *)
						ePath := PATH_GENERIC, bExecute := TRUE );
		step := 2;

	2:(* Wait until open not busy *)
		fbFileOpen( bExecute := FALSE, bError => bError, nErrID => nErrID, hFile => hFile );
		IF NOT fbFileOpen.bBusy THEN
			IF NOT fbFileOpen.bError THEN
				step := 3;
			ELSE(* Error: file not found? *)
				step := 100;
			END_IF
		END_IF
		
	3:(* Convert one PLC record to CSV format *)
		sCSVLine := '';
		fbWriter.eCmd := eEnumCmd_First;(* Write first field value *)
		
		FOR nColumn := 1 TO MAX_CSV_COLUMNS BY 1 DO
				
				IF nColumn = 1 THEN
					sCSVField := STRING_TO_CSVFIELD(sColumn1TimeStamp, FALSE);
				ELSIF nColumn = 2 THEN
					sCSVField := STRING_TO_CSVFIELD(sColumn2, FALSE);
				ELSIF nColumn = 3 THEN
					sCSVField := STRING_TO_CSVFIELD(sColumn3, FALSE);
				ELSIF nColumn = 4 THEN
					sCSVField := STRING_TO_CSVFIELD(sColumn4, FALSE);
				ELSIF nColumn = 5 THEN
					sCSVField := STRING_TO_CSVFIELD(sColumn5, FALSE);
				ELSIF nColumn = 6 THEN	
					sCSVField := STRING_TO_CSVFIELD(sColumn6, FALSE);
				ELSIF nColumn = 7 THEN	
					sCSVField := STRING_TO_CSVFIELD(sColumn7, FALSE);
				END_IF
				
				(* Add new field to the record buffer *)
				fbWriter( 	pBuffer := ADR( sCSVLine ), cbBuffer := SIZEOF( sCSVLine ) - 1, putValue := sCSVField, pValue := 0, cbValue := 0,
							bCRLF := ( nColumn = MAX_CSV_COLUMNS ) );
										
				IF fbWriter.bOk THEN
					fbWriter.eCmd := eEnumCmd_Next;(* Write next field value *)
				ELSE(* Error *)
					step := 100;
					RETURN;
				END_IF

		END_FOR

		(* FB_FilePuts adds allready CR (carriage return) to the written line.
		We have to replace the $R$L characters with $L character to avoid double CR. *)
		IF RIGHT( sCSVLine, 2 ) = '$R$L' THEN
			sCSVLine := REPLACE( sCSVLine, '$L', 2, LEN( sCSVLine ) - 1 );
		END_IF

		step := 4;(* Write record to the file *)
		
	4:	(* Write single text line *)
		fbFilePuts( bExecute := FALSE );
		fbFilePuts( sNetId := sNetId, hFile := hFile, sLine := sCSVLine, bExecute := TRUE );
		step := 5;

	5:(* Wait until write not busy *)
		fbFilePuts( bExecute := FALSE, bError => bError, nErrID => nErrID );
		IF NOT fbFilePuts.bBusy THEN
			IF NOT fbFilePuts.bError THEN
				step := 10;(* Close file *)
			ELSE(* Error *)
				step := 100;
			END_IF
		END_IF

	10:	(* Close source file *)
		fbFileClose( bExecute := FALSE );
		fbFileClose( sNetId := sNetId, hFile := hFile, bExecute := TRUE );
		step := 11;

	11:(* Wait until close not busy *)
		fbFileClose( bExecute := FALSE, bError => bError, nErrID => nErrID );
		IF ( NOT fbFileClose.bBusy ) THEN
			hFile := 0;
			step := 100;
		END_IF

	100: (* Error or ready step => cleanup *)
		IF ( hFile <> 0 ) THEN
			step := 10; (* Close the source file *)
		ELSE
			bBusy := FALSE;
			step := 0;	(* Ready *)
		END_IF

END_CASE

END_FUNCTION_BLOCK

// ---- POUs/Loggning/Cluster_Logg.TcPOU
PROGRAM Cluster_Logg
VAR
	
fbLogg1 		:FB_SaveToCSV_ClusterCtrl;
	tUpdateTime1	:TIME:=T#5S;
	sFileName1		:STRING(255):='Unit1_1';
	
	fbLogg2 		:FB_SaveToCSV_ClusterCtrl;
	tUpdateTime2	:TIME:=T#5S;
	sFileName2		:STRING(255):='Unit1_2';
	
	fbLogg3 		:FB_SaveToCSV_ClusterCtrl;
	tUpdateTime3	:TIME:=T#5S;
	sFileName3		:STRING(255):='Unit1_3';
	
END_VAR

fbLogg1(
	bChangeSeparatorToComma:= FALSE, 
	bExecute:= GVL_Fastighet.CSVClusterCtrl, 
	tUpdateTime:= tUpdateTime1, 
	sFileName:= sFileName1, 
	nDayOfWeek:= PLC_TID.fbTime.systemTime.wDayOfWeek,
	sColumn1TimeStamp:= PLC_TID.systemTime, 
	sColumn2:= REAL_TO_STRING(GVL_ClusterCtrl._CCtrl_V1_P1), 
	sColumn3:= REAL_TO_STRING(GVL_ClusterCtrl._CCtrl_V1_P2), 
	sColumn4:= REAL_TO_STRING(GVL_ClusterCtrl._CCtrl_V1_P3), 
	sColumn5:= REAL_TO_STRING(GVL_ClusterCtrl._CCtrl_V1_U1_L1_N), 
	sColumn6:= REAL_TO_STRING(GVL_ClusterCtrl._CCtrl_V1_U2_L2_N), 
	sColumn7:= REAL_TO_STRING(GVL_ClusterCtrl._CCtrl_V1_U3_L3_N),
	sColumn8:= REAL_TO_STRING(GVL_ClusterCtrl._CCtrl_V1_HZ));
	
	fbLogg2(
	bChangeSeparatorToComma:= FALSE, 
	bExecute:= GVL_Fastighet.CSVClusterCtrl, 
	tUpdateTime:= tUpdateTime2, 
	sFileName:= sFileName2, 
	nDayOfWeek:= PLC_TID.fbTime.systemTime.wDayOfWeek,
	sColumn1TimeStamp:= PLC_TID.systemTime, 
	sColumn2:= REAL_TO_STRING(GVL_ClusterCtrl._CCtrl_V1_U1_L1_L2), 
	sColumn3:= REAL_TO_STRING(GVL_ClusterCtrl._CCtrl_V1_U2_L2_L3), 
	sColumn4:= REAL_TO_STRING(GVL_ClusterCtrl._CCtrl_V1_U3_L3_L1), 
	sColumn5:= REAL_TO_STRING(GVL_ClusterCtrl._CCtrl_V1_Itot),
	sColumn6:= REAL_TO_STRING(GVL_ClusterCtrl._CCtrl_V1_I1), 
	sColumn7:= REAL_TO_STRING(GVL_ClusterCtrl._CCtrl_V1_I2), 
	sColumn8:= REAL_TO_STRING(GVL_ClusterCtrl._CCtrl_V1_I3));
	
	fbLogg3(
	bChangeSeparatorToComma:= FALSE, 
	bExecute:= GVL_Fastighet.CSVClusterCtrl, 
	tUpdateTime:= tUpdateTime3, 
	sFileName:= sFileName3, 
	nDayOfWeek:= PLC_TID.fbTime.systemTime.wDayOfWeek,
	sColumn1TimeStamp:= PLC_TID.systemTime, 
	sColumn2:= REAL_TO_STRING(GVL_ClusterCtrl._CCtrl_V1_Yield_Wh), 
	sColumn3:= REAL_TO_STRING(GVL_ClusterCtrl._CCtrl_V1_Yield_kWh), 
	sColumn4:= REAL_TO_STRING(GVL_ClusterCtrl._CCtrl_V1_Yield_MWh), 
	sColumn5:= REAL_TO_STRING(GVL_ClusterCtrl._CCtrl_V1_YieldDay_Wh), 
	sColumn6:= REAL_TO_STRING(GVL_ClusterCtrl._CCtrl_V1_YieldDay_kWh), 
	sColumn7:= REAL_TO_STRING(GVL_ClusterCtrl._CCtrl_V1_P));

END_PROGRAM

// ---- POUs/_FBs/FB_SaveToCSV_ClusterCtrl.TcPOU
FUNCTION_BLOCK FB_SaveToCSV_ClusterCtrl
VAR CONSTANT
	MAX_CSV_COLUMNS 	: UDINT := 8;
END_VAR
VAR_INPUT
	(*	In USA/UK the CSV field separator is a comma.
	In Germany and some other European countries the CSV field separator is a semicolon. *)
	bChangeSeparatorToComma	: BOOL := FALSE;
	bExecute : BOOL;
	tUpdateTime : TIME:=T#1S; //Update time 
	sFileName	: T_MaxString := 'DefaultName';(* CSV destination file path and name *)
	nDayOfWeek : WORD;
	sColumn1TimeStamp : T_MaxString;
	sColumn2 : STRING;
	sColumn3 : STRING;
	sColumn4 : STRING; 
	sColumn5 : STRING;
	sColumn6 : STRING;
	sColumn7 : STRING;
	sColumn8 : STRING;
END_VAR
VAR
	sNetId			: T_AmsNetId := '';	(* TwinCAT system network address *)	
	sCSVLine		: T_MaxString := '';(* Single CSV text line (row, record), we are using string as record buffer (your are able to see created fields) *)
	sCSVField		: T_MaxString := '';(* Single CSV field value (column, record field) *)
	bBusy			: BOOL;
	bError			: BOOL;
	nErrId			: UDINT;
	nColumn		: UDINT 	:= 1;(* Column number (record field) *)
	hFile			: UINT		:= 0;(* File handle of the source file *)
	step			: DWORD 	:= 0;
	fbFileOpen	: FB_FileOpen;(* Opens file *)
	fbFileClose	: FB_FileClose;(* Closes file *)
	fbFilePuts		: FB_FilePuts;(* Writes one record (line) *)
	fbWriter		: FB_CSVMemBufferWriter;(* Helper function block used to create CSV data bytes (single record line) *)	
	tUpdateTimer : TON;
	sCompleteFileName : STRING;
	sPathName : T_MaxString;
	sTempDate : STRING;
	sDate : STRING;
	bWeekUpdate : BOOL;
END_VAR

(* Call the timer every plc-cycle *)
tUpdateTimer(IN:=NOT tUpdateTimer.Q, PT:=tUpdateTime);


(* Update filename *)
IF nDayOfWeek = 1 AND bWeekUpdate THEN //1=Monday	
		sCompleteFileName	:= sFileName;
		sTempDate := DELETE(sColumn1TimeStamp, 16,11); //Cut the timestamp so we only save the date
		sDate := INSERT(sTempDate, '_', 10); //Add '-' after the date for seperation
		sPathName:=CONCAT(CONCAT('C:\Loggning\Cluster\',CONCAT(sDate,sFileName)),'.csv');
		bWeekUpdate := FALSE;
ELSE
	(* Update if name has changed *)
	IF sCompleteFileName <> sFileName THEN
		sCompleteFileName := sFileName;
		sTempDate := DELETE(sColumn1TimeStamp, 16,11); //Cut the timestamp so we only save the date
		sDate := INSERT(sTempDate, '_', 10); //Add '-' after the date for seperation
		sPathName:=CONCAT(CONCAT('C:\Loggning\Cluster\',CONCAT(sDate,sCompleteFileName)),'.csv');
	END_IF	
END_IF

IF nDayOfWeek <> 1 THEN
	bWeekUpdate := TRUE;
END_IF

CASE step OF
	0:	(* Wait for rising edge at bWrite variable *)
		IF bExecute AND tUpdateTimer.Q THEN
			bBusy 		:= TRUE;
			bError		:= FALSE;
			nErrId		:= 0;
			hFile			:= 0;
			step 		:= 1;
		END_IF

	1:	(* Open source file *)
		fbFileOpen(  bExecute := FALSE  );
		fbFileOpen( 	sNetId := sNetId, sPathName := sPathName, nMode := FOPEN_MODEAPPEND OR FOPEN_MODETEXT,(* Open file in TEXT mode! *)
						ePath := PATH_GENERIC, bExecute := TRUE );
		step := 2;

	2:(* Wait until open not busy *)
		fbFileOpen( bExecute := FALSE, bError => bError, nErrID => nErrID, hFile => hFile );
		IF NOT fbFileOpen.bBusy THEN
			IF NOT fbFileOpen.bError THEN
				step := 3;
			ELSE(* Error: file not found? *)
				step := 100;
			END_IF
		END_IF
		
	3:(* Convert one PLC record to CSV format *)
		sCSVLine := '';
		fbWriter.eCmd := eEnumCmd_First;(* Write first field value *)
		
		FOR nColumn := 1 TO MAX_CSV_COLUMNS BY 1 DO
				
				IF nColumn = 1 THEN
					sCSVField := STRING_TO_CSVFIELD(sColumn1TimeStamp, FALSE);
				ELSIF nColumn = 2 THEN
					sCSVField := STRING_TO_CSVFIELD(sColumn2, FALSE);
				ELSIF nColumn = 3 THEN
					sCSVField := STRING_TO_CSVFIELD(sColumn3, FALSE);
				ELSIF nColumn = 4 THEN
					sCSVField := STRING_TO_CSVFIELD(sColumn4, FALSE);
				ELSIF nColumn = 5 THEN
					sCSVField := STRING_TO_CSVFIELD(sColumn5, FALSE);
				ELSIF nColumn = 6 THEN	
					sCSVField := STRING_TO_CSVFIELD(sColumn6, FALSE);
				ELSIF nColumn = 7 THEN	
					sCSVField := STRING_TO_CSVFIELD(sColumn7, FALSE);
				ELSIF nColumn = 8 THEN	
					sCSVField := STRING_TO_CSVFIELD(sColumn8, FALSE);
				END_IF
				
				(* Add new field to the record buffer *)
				fbWriter( 	pBuffer := ADR( sCSVLine ), cbBuffer := SIZEOF( sCSVLine ) - 1, putValue := sCSVField, pValue := 0, cbValue := 0,
							bCRLF := ( nColumn = MAX_CSV_COLUMNS ) );
										
				IF fbWriter.bOk THEN
					fbWriter.eCmd := eEnumCmd_Next;(* Write next field value *)
				ELSE(* Error *)
					step := 100;
					RETURN;
				END_IF

		END_FOR

		(* FB_FilePuts adds allready CR (carriage return) to the written line.
		We have to replace the $R$L characters with $L character to avoid double CR. *)
		IF RIGHT( sCSVLine, 2 ) = '$R$L' THEN
			sCSVLine := REPLACE( sCSVLine, '$L', 2, LEN( sCSVLine ) - 1 );
		END_IF

		step := 4;(* Write record to the file *)
		
	4:	(* Write single text line *)
		fbFilePuts( bExecute := FALSE );
		fbFilePuts( sNetId := sNetId, hFile := hFile, sLine := sCSVLine, bExecute := TRUE );
		step := 5;

	5:(* Wait until write not busy *)
		fbFilePuts( bExecute := FALSE, bError => bError, nErrID => nErrID );
		IF NOT fbFilePuts.bBusy THEN
			IF NOT fbFilePuts.bError THEN
				step := 10;(* Close file *)
			ELSE(* Error *)
				step := 100;
			END_IF
		END_IF

	10:	(* Close source file *)
		fbFileClose( bExecute := FALSE );
		fbFileClose( sNetId := sNetId, hFile := hFile, bExecute := TRUE );
		step := 11;

	11:(* Wait until close not busy *)
		fbFileClose( bExecute := FALSE, bError => bError, nErrID => nErrID );
		IF ( NOT fbFileClose.bBusy ) THEN
			hFile := 0;
			step := 100;
		END_IF

	100: (* Error or ready step => cleanup *)
		IF ( hFile <> 0 ) THEN
			step := 10; (* Close the source file *)
		ELSE
			bBusy := FALSE;
			step := 0;	(* Ready *)
		END_IF

END_CASE

END_FUNCTION_BLOCK

// ---- POUs/Loggning/Cluster_Logg_2.TcPOU
PROGRAM Cluster_Logg_2
VAR
	
	fbLogg1 		:FB_SaveToCSV_ClusterCtrl;
	tUpdateTime1	:TIME:=T#5S;
	sFileName1		:STRING(255):='Unit2_1';
	
	fbLogg2 		:FB_SaveToCSV_ClusterCtrl;
	tUpdateTime2	:TIME:=T#5S;
	sFileName2		:STRING(255):='Unit2_2';
	
	fbLogg3 		:FB_SaveToCSV_ClusterCtrl;
	tUpdateTime3	:TIME:=T#5S;
	sFileName3		:STRING(255):='Unit2_3';
	
END_VAR

fbLogg1(	
	bChangeSeparatorToComma:= FALSE, 
	bExecute:= GVL_Fastighet.CSVClusterCtrl, 
	tUpdateTime:= tUpdateTime1, 
	sFileName:= sFileName1, 
	nDayOfWeek:= PLC_TID.fbTime.systemTime.wDayOfWeek,
	sColumn1TimeStamp:= PLC_TID.systemTime, 
	sColumn2:= REAL_TO_STRING(GVL_ClusterCtrl._CCtrl_V2_P1), 
	sColumn3:= REAL_TO_STRING(GVL_ClusterCtrl._CCtrl_V2_P2), 
	sColumn4:= REAL_TO_STRING(GVL_ClusterCtrl._CCtrl_V2_P3), 
	sColumn5:= REAL_TO_STRING(GVL_ClusterCtrl._CCtrl_V2_U1_L1_N), 
	sColumn6:= REAL_TO_STRING(GVL_ClusterCtrl._CCtrl_V2_U2_L2_N), 
	sColumn7:= REAL_TO_STRING(GVL_ClusterCtrl._CCtrl_V2_U3_L3_N),
	sColumn8:= REAL_TO_STRING(GVL_ClusterCtrl._CCtrl_V2_HZ));
	
	fbLogg2(
	bChangeSeparatorToComma:= FALSE, 
	bExecute:= GVL_Fastighet.CSVClusterCtrl, 
	tUpdateTime:= tUpdateTime2, 
	sFileName:= sFileName2, 
	nDayOfWeek:= PLC_TID.fbTime.systemTime.wDayOfWeek,
	sColumn1TimeStamp:= PLC_TID.systemTime, 
	sColumn2:= REAL_TO_STRING(GVL_ClusterCtrl._CCtrl_V2_U1_L1_L2), 
	sColumn3:= REAL_TO_STRING(GVL_ClusterCtrl._CCtrl_V2_U2_L2_L3), 
	sColumn4:= REAL_TO_STRING(GVL_ClusterCtrl._CCtrl_V2_U3_L3_L1), 
	sColumn5:= REAL_TO_STRING(GVL_ClusterCtrl._CCtrl_V2_Itot), 
	sColumn6:= REAL_TO_STRING(GVL_ClusterCtrl._CCtrl_V2_I1), 
	sColumn7:= REAL_TO_STRING(GVL_ClusterCtrl._CCtrl_V2_I2), 
	sColumn8:= REAL_TO_STRING(GVL_ClusterCtrl._CCtrl_V2_I3));
	
	fbLogg3(
	bChangeSeparatorToComma:= FALSE, 
	bExecute:= GVL_Fastighet.CSVClusterCtrl, 
	tUpdateTime:= tUpdateTime3, 
	sFileName:= sFileName3, 
	nDayOfWeek:= PLC_TID.fbTime.systemTime.wDayOfWeek,
	sColumn1TimeStamp:= PLC_TID.systemTime, 
	sColumn2:= REAL_TO_STRING(GVL_ClusterCtrl._CCtrl_V2_Yield_Wh), 
	sColumn3:= REAL_TO_STRING(GVL_ClusterCtrl._CCtrl_V2_Yield_kWh), 
	sColumn4:= REAL_TO_STRING(GVL_ClusterCtrl._CCtrl_V2_Yield_MWh), 
	sColumn5:= REAL_TO_STRING(GVL_ClusterCtrl._CCtrl_V2_YieldDay_Wh), 
	sColumn6:= REAL_TO_STRING(GVL_ClusterCtrl._CCtrl_V2_YieldDay_kWh), 
	sColumn7:= REAL_TO_STRING(GVL_ClusterCtrl._CCtrl_V2_P));

END_PROGRAM

// ---- POUs/Loggning/Cluster_Logg_3.TcPOU
PROGRAM Cluster_Logg_3
VAR
	
	fbLogg1 		:FB_SaveToCSV_ClusterCtrl;
	tUpdateTime1	:TIME:=T#5S;
	sFileName1		:STRING(255):='Unit3_1';
	
	fbLogg2 		:FB_SaveToCSV_ClusterCtrl;
	tUpdateTime2	:TIME:=T#5S;
	sFileName2		:STRING(255):='Unit3_2';
	
	fbLogg3 		:FB_SaveToCSV_ClusterCtrl;
	tUpdateTime3	:TIME:=T#5S;
	sFileName3		:STRING(255):='Unit3_3';
	


END_VAR

fbLogg1(	
	bChangeSeparatorToComma:= FALSE, 
	bExecute:= GVL_Fastighet.CSVClusterCtrl, 
	tUpdateTime:= tUpdateTime1, 
	sFileName:= sFileName1, 
	nDayOfWeek:= PLC_TID.fbTime.systemTime.wDayOfWeek,
	sColumn1TimeStamp:= PLC_TID.systemTime, 
	sColumn2:= REAL_TO_STRING(GVL_ClusterCtrl._CCtrl_V3_P1), 
	sColumn3:= REAL_TO_STRING(GVL_ClusterCtrl._CCtrl_V3_P2), 
	sColumn4:= REAL_TO_STRING(GVL_ClusterCtrl._CCtrl_V3_P3), 
	sColumn5:= REAL_TO_STRING(GVL_ClusterCtrl._CCtrl_V3_U1_L1_N), 
	sColumn6:= REAL_TO_STRING(GVL_ClusterCtrl._CCtrl_V3_U2_L2_N), 
	sColumn7:= REAL_TO_STRING(GVL_ClusterCtrl._CCtrl_V3_U3_L3_N),
	sColumn8:= REAL_TO_STRING(GVL_ClusterCtrl._CCtrl_V3_HZ));
	
	fbLogg2(
	bChangeSeparatorToComma:= FALSE, 
	bExecute:= GVL_Fastighet.CSVClusterCtrl, 
	tUpdateTime:= tUpdateTime2, 
	sFileName:= sFileName2, 
	nDayOfWeek:= PLC_TID.fbTime.systemTime.wDayOfWeek,
	sColumn1TimeStamp:= PLC_TID.systemTime, 
	sColumn2:= REAL_TO_STRING(GVL_ClusterCtrl._CCtrl_V3_U1_L1_L2), 
	sColumn3:= REAL_TO_STRING(GVL_ClusterCtrl._CCtrl_V3_U2_L2_L3), 
	sColumn4:= REAL_TO_STRING(GVL_ClusterCtrl._CCtrl_V3_U3_L3_L1), 
	sColumn5:= REAL_TO_STRING(GVL_ClusterCtrl._CCtrl_V3_Itot), 
	sColumn6:= REAL_TO_STRING(GVL_ClusterCtrl._CCtrl_V3_I1), 
	sColumn7:= REAL_TO_STRING(GVL_ClusterCtrl._CCtrl_V3_I2), 
	sColumn8:= REAL_TO_STRING(GVL_ClusterCtrl._CCtrl_V3_I3));
	
	fbLogg3(
	bChangeSeparatorToComma:= FALSE, 
	bExecute:= GVL_Fastighet.CSVClusterCtrl, 
	tUpdateTime:= tUpdateTime3, 
	sFileName:= sFileName3, 
	nDayOfWeek:= PLC_TID.fbTime.systemTime.wDayOfWeek,
	sColumn1TimeStamp:= PLC_TID.systemTime, 
	sColumn2:= REAL_TO_STRING(GVL_ClusterCtrl._CCtrl_V3_Yield_Wh), 
	sColumn3:= REAL_TO_STRING(GVL_ClusterCtrl._CCtrl_V3_Yield_kWh), 
	sColumn4:= REAL_TO_STRING(GVL_ClusterCtrl._CCtrl_V3_Yield_MWh), 
	sColumn5:= REAL_TO_STRING(GVL_ClusterCtrl._CCtrl_V3_YieldDay_Wh), 
	sColumn6:= REAL_TO_STRING(GVL_ClusterCtrl._CCtrl_V3_YieldDay_kWh), 
	sColumn7:= REAL_TO_STRING(GVL_ClusterCtrl._CCtrl_V3_P));

END_PROGRAM

// ---- POUs/Loggning/Cluster_Sensor_Logg.TcPOU
PROGRAM Cluster_Sensor_Logg
VAR
	
	fbLogg1 		:FB_SaveToCSV_Cluster_Sensors;
	tUpdateTime1	:TIME:=T#5S;
	sFileName1		:STRING(255):='Sensor_Logg';
	
	

END_VAR

fbLogg1(
	bChangeSeparatorToComma:= FALSE, 
	bExecute:= GVL_Fastighet.CSVClusterCtrl, 
	tUpdateTime:= tUpdateTime1, 
	sFileName:= sFileName1, 
	nDayOfWeek:= PLC_TID.fbTime.systemTime.wDayOfWeek,
	sColumn1TimeStamp:= PLC_TID.systemTime, 
	sColumn2:= REAL_TO_STRING(GVL_ClusterCtrl._CCtrl_ST_Si420TC), );

END_PROGRAM

// ---- POUs/_FBs/FB_SaveToCSV_Cluster_Sensors.TcPOU
FUNCTION_BLOCK FB_SaveToCSV_Cluster_Sensors
VAR CONSTANT
	MAX_CSV_COLUMNS 	: UDINT := 2;
END_VAR
VAR_INPUT
	(*	In USA/UK the CSV field separator is a comma.
	In Germany and some other European countries the CSV field separator is a semicolon. *)
	bChangeSeparatorToComma	: BOOL := FALSE;
	bExecute : BOOL;
	tUpdateTime : TIME:=T#5S; //Update time 
	sFileName	: T_MaxString := 'Sensor_Logg';(* CSV destination file path and name *)
	nDayOfWeek : WORD;
	sColumn1TimeStamp : T_MaxString;
	sColumn2 : STRING;
END_VAR
VAR
	sNetId			: T_AmsNetId := '';	(* TwinCAT system network address *)	
	sCSVLine		: T_MaxString := '';(* Single CSV text line (row, record), we are using string as record buffer (your are able to see created fields) *)
	sCSVField		: T_MaxString := '';(* Single CSV field value (column, record field) *)
	bBusy			: BOOL;
	bError			: BOOL;
	nErrId			: UDINT;
	nColumn		: UDINT 	:= 1;(* Column number (record field) *)
	hFile			: UINT		:= 0;(* File handle of the source file *)
	step			: DWORD 	:= 0;
	fbFileOpen	: FB_FileOpen;(* Opens file *)
	fbFileClose	: FB_FileClose;(* Closes file *)
	fbFilePuts		: FB_FilePuts;(* Writes one record (line) *)
	fbWriter		: FB_CSVMemBufferWriter;(* Helper function block used to create CSV data bytes (single record line) *)	
	tUpdateTimer : TON;
	sCompleteFileName : STRING;
	sPathName : T_MaxString;
	sTempDate : STRING;
	sDate : STRING;
	bWeekUpdate : BOOL;
END_VAR

(* Call the timer every plc-cycle *)
tUpdateTimer(IN:=NOT tUpdateTimer.Q, PT:=tUpdateTime);


(* Update filename *)
IF nDayOfWeek = 1 AND bWeekUpdate THEN //1=Monday	
		sCompleteFileName	:= sFileName;
		sTempDate := DELETE(sColumn1TimeStamp, 16,11); //Cut the timestamp so we only save the date
		sDate := INSERT(sTempDate, '_', 10); //Add '-' after the date for seperation
		sPathName:=CONCAT(CONCAT('C:\Loggning\Sensor_Logg\',CONCAT(sDate,sFileName)),'.csv');
		bWeekUpdate := FALSE;
ELSE
	(* Update if name has changed *)
	IF sCompleteFileName <> sFileName THEN
		sCompleteFileName := sFileName;
		sTempDate := DELETE(sColumn1TimeStamp, 16,11); //Cut the timestamp so we only save the date
		sDate := INSERT(sTempDate, '_', 10); //Add '-' after the date for seperation
		sPathName:=CONCAT(CONCAT('C:\Loggning\Sensor_Logg\',CONCAT(sDate,sCompleteFileName)),'.csv');
	END_IF	
END_IF

IF nDayOfWeek <> 1 THEN
	bWeekUpdate := TRUE;
END_IF

CASE step OF
	0:	(* Wait for rising edge at bWrite variable *)
		IF bExecute AND tUpdateTimer.Q THEN
			bBusy 		:= TRUE;
			bError		:= FALSE;
			nErrId		:= 0;
			hFile			:= 0;
			step 		:= 1;
		END_IF

	1:	(* Open source file *)
		fbFileOpen(  bExecute := FALSE  );
		fbFileOpen( 	sNetId := sNetId, sPathName := sPathName, nMode := FOPEN_MODEAPPEND OR FOPEN_MODETEXT,(* Open file in TEXT mode! *)
						ePath := PATH_GENERIC, bExecute := TRUE );
		step := 2;

	2:(* Wait until open not busy *)
		fbFileOpen( bExecute := FALSE, bError => bError, nErrID => nErrID, hFile => hFile );
		IF NOT fbFileOpen.bBusy THEN
			IF NOT fbFileOpen.bError THEN
				step := 3;
			ELSE(* Error: file not found? *)
				step := 100;
			END_IF
		END_IF
		
	3:(* Convert one PLC record to CSV format *)
		sCSVLine := '';
		fbWriter.eCmd := eEnumCmd_First;(* Write first field value *)
		
		FOR nColumn := 1 TO MAX_CSV_COLUMNS BY 1 DO
				
				IF nColumn = 1 THEN
					sCSVField := STRING_TO_CSVFIELD(sColumn1TimeStamp, FALSE);
				ELSIF nColumn = 2 THEN
					sCSVField := STRING_TO_CSVFIELD(sColumn2, FALSE);
				END_IF
				
				(* Add new field to the record buffer *)
				fbWriter( 	pBuffer := ADR( sCSVLine ), cbBuffer := SIZEOF( sCSVLine ) - 1, putValue := sCSVField, pValue := 0, cbValue := 0,
							bCRLF := ( nColumn = MAX_CSV_COLUMNS ) );
										
				IF fbWriter.bOk THEN
					fbWriter.eCmd := eEnumCmd_Next;(* Write next field value *)
				ELSE(* Error *)
					step := 100;
					RETURN;
				END_IF

		END_FOR

		(* FB_FilePuts adds allready CR (carriage return) to the written line.
		We have to replace the $R$L characters with $L character to avoid double CR. *)
		IF RIGHT( sCSVLine, 2 ) = '$R$L' THEN
			sCSVLine := REPLACE( sCSVLine, '$L', 2, LEN( sCSVLine ) - 1 );
		END_IF

		step := 4;(* Write record to the file *)
		
	4:	(* Write single text line *)
		fbFilePuts( bExecute := FALSE );
		fbFilePuts( sNetId := sNetId, hFile := hFile, sLine := sCSVLine, bExecute := TRUE );
		step := 5;

	5:(* Wait until write not busy *)
		fbFilePuts( bExecute := FALSE, bError => bError, nErrID => nErrID );
		IF NOT fbFilePuts.bBusy THEN
			IF NOT fbFilePuts.bError THEN
				step := 10;(* Close file *)
			ELSE(* Error *)
				step := 100;
			END_IF
		END_IF

	10:	(* Close source file *)
		fbFileClose( bExecute := FALSE );
		fbFileClose( sNetId := sNetId, hFile := hFile, bExecute := TRUE );
		step := 11;

	11:(* Wait until close not busy *)
		fbFileClose( bExecute := FALSE, bError => bError, nErrID => nErrID );
		IF ( NOT fbFileClose.bBusy ) THEN
			hFile := 0;
			step := 100;
		END_IF

	100: (* Error or ready step => cleanup *)
		IF ( hFile <> 0 ) THEN
			step := 10; (* Close the source file *)
		ELSE
			bBusy := FALSE;
			step := 0;	(* Ready *)
		END_IF

END_CASE

END_FUNCTION_BLOCK

// ---- POUs/Loggning/WXT530_Logg.TcPOU
PROGRAM WXT530_Logg
VAR
	
	fbLogg1 		:FB_SaveToCSV_WXT530;
	tUpdateTime1	:TIME:=T#5S;
	sFileName1		:STRING(255):='WXT5301';
	
	fbLogg2 		:FB_SaveToCSV_WXT530;
	tUpdateTime2	:TIME:=T#5S;
	sFileName2		:STRING(255):='WXT5302';
	
	fbLogg3 		:FB_SaveToCSV_WXT530;
	tUpdateTime3	:TIME:=T#5S;
	sFileName3		:STRING(255):='WXT5303';
	
END_VAR

fbLogg1(
	bChangeSeparatorToComma:= FALSE, 
	bExecute:= GVL_Fastighet.CSVWXT530, 
	tUpdateTime:= tUpdateTime1, 
	sFileName:= sFileName1, 
	nDayOfWeek:= PLC_TID.fbTime.systemTime.wDayOfWeek,
	sColumn1TimeStamp:= PLC_TID.systemTime, 
	sColumn2:= REAL_TO_STRING(GVL_WXT530._GW3U_DN), 
	sColumn3:= REAL_TO_STRING(GVL_WXT530._GW3U_DM), 
	sColumn4:= REAL_TO_STRING(GVL_WXT530._GW3U_DX), 
	sColumn5:= REAL_TO_STRING(GVL_WXT530._GW3U_SN), 
	sColumn6:= REAL_TO_STRING(GVL_WXT530._GW3U_SM), 
	sColumn7:= REAL_TO_STRING(GVL_WXT530._GW3U_SX));
	
	
fbLogg2(
	bChangeSeparatorToComma:= FALSE, 
	bExecute:= GVL_Fastighet.CSVWXT530, 
	tUpdateTime:= tUpdateTime2, 
	sFileName:= sFileName2, 
	nDayOfWeek:= PLC_TID.fbTime.systemTime.wDayOfWeek,
	sColumn1TimeStamp:= PLC_TID.systemTime, 
	sColumn2:= REAL_TO_STRING(GVL_WXT530._GW3U_GT3U), 
	sColumn3:= REAL_TO_STRING(GVL_WXT530._GW3U_GT41), 
	sColumn4:= REAL_TO_STRING(GVL_WXT530._GW3U_GM41), 
	sColumn5:= REAL_TO_STRING(GVL_WXT530._GW3U_GP41), 
	sColumn6:= REAL_TO_STRING(GVL_WXT530._GW3U_RC), 
	sColumn7:= REAL_TO_STRING(GVL_WXT530._GW3U_RD));
	
	
	fbLogg3(
	bChangeSeparatorToComma:= FALSE, 
	bExecute:= GVL_Fastighet.CSVWXT530, 
	tUpdateTime:= tUpdateTime3, 
	sFileName:= sFileName3, 
	nDayOfWeek:= PLC_TID.fbTime.systemTime.wDayOfWeek,
	sColumn1TimeStamp:= PLC_TID.systemTime, 
	sColumn2:= REAL_TO_STRING(GVL_WXT530._GW3U_RI), 
	sColumn3:= REAL_TO_STRING(GVL_WXT530._GW3U_HC), 
	sColumn4:= REAL_TO_STRING(GVL_WXT530._GW3U_HD), 
	sColumn5:= REAL_TO_STRING(GVL_WXT530._GW3U_HI), 
	sColumn6:= REAL_TO_STRING(GVL_WXT530._GW3U_RP), 
	sColumn7:= REAL_TO_STRING(GVL_WXT530._GW3U_HP));

END_PROGRAM

// ---- POUs/_FBs/FB_SaveToCSV_WXT530.TcPOU
FUNCTION_BLOCK FB_SaveToCSV_WXT530
VAR CONSTANT
	MAX_CSV_COLUMNS 	: UDINT := 7;
END_VAR
VAR_INPUT
	(*	In USA/UK the CSV field separator is a comma.
	In Germany and some other European countries the CSV field separator is a semicolon. *)
	bChangeSeparatorToComma	: BOOL := FALSE;
	bExecute : BOOL;
	tUpdateTime : TIME:=T#1S; //Update time 
	sFileName	: T_MaxString := 'DefaultName';(* CSV destination file path and name *)
	nDayOfWeek : WORD;
	sColumn1TimeStamp : T_MaxString;
	sColumn2 : STRING;
	sColumn3 : STRING;
	sColumn4 : STRING; 
	sColumn5 : STRING;
	sColumn6 : STRING;
	sColumn7 : STRING;
END_VAR
VAR
	sNetId			: T_AmsNetId := '';	(* TwinCAT system network address *)	
	sCSVLine		: T_MaxString := '';(* Single CSV text line (row, record), we are using string as record buffer (your are able to see created fields) *)
	sCSVField		: T_MaxString := '';(* Single CSV field value (column, record field) *)
	bBusy			: BOOL;
	bError			: BOOL;
	nErrId			: UDINT;
	nColumn		: UDINT 	:= 1;(* Column number (record field) *)
	hFile			: UINT		:= 0;(* File handle of the source file *)
	step			: DWORD 	:= 0;
	fbFileOpen	: FB_FileOpen;(* Opens file *)
	fbFileClose	: FB_FileClose;(* Closes file *)
	fbFilePuts		: FB_FilePuts;(* Writes one record (line) *)
	fbWriter		: FB_CSVMemBufferWriter;(* Helper function block used to create CSV data bytes (single record line) *)	
	tUpdateTimer : TON;
	sCompleteFileName : STRING;
	sPathName : T_MaxString;
	sTempDate : STRING;
	sDate : STRING;
	bWeekUpdate : BOOL;
END_VAR

(* Call the timer every plc-cycle *)
tUpdateTimer(IN:=NOT tUpdateTimer.Q, PT:=tUpdateTime);


(* Update filename *)
IF nDayOfWeek = 1 AND bWeekUpdate THEN //1=Monday	
		sCompleteFileName	:= sFileName;
		sTempDate := DELETE(sColumn1TimeStamp, 16,11); //Cut the timestamp so we only save the date
		sDate := INSERT(sTempDate, '_', 10); //Add '-' after the date for seperation
		sPathName:=CONCAT(CONCAT('C:\Loggning\Vader\',CONCAT(sDate,sFileName)),'.csv');
		bWeekUpdate := FALSE;
ELSE
	(* Update if name has changed *)
	IF sCompleteFileName <> sFileName THEN
		sCompleteFileName := sFileName;
		sTempDate := DELETE(sColumn1TimeStamp, 16,11); //Cut the timestamp so we only save the date
		sDate := INSERT(sTempDate, '_', 10); //Add '-' after the date for seperation
		sPathName:=CONCAT(CONCAT('C:\Loggning\Vader\',CONCAT(sDate,sCompleteFileName)),'.csv');
	END_IF	
END_IF

IF nDayOfWeek <> 1 THEN
	bWeekUpdate := TRUE;
END_IF

CASE step OF
	0:	(* Wait for rising edge at bWrite variable *)
		IF bExecute AND tUpdateTimer.Q THEN
			bBusy 		:= TRUE;
			bError		:= FALSE;
			nErrId		:= 0;
			hFile			:= 0;
			step 		:= 1;
		END_IF

	1:	(* Open source file *)
		fbFileOpen(  bExecute := FALSE  );
		fbFileOpen( 	sNetId := sNetId, sPathName := sPathName, nMode := FOPEN_MODEAPPEND OR FOPEN_MODETEXT,(* Open file in TEXT mode! *)
						ePath := PATH_GENERIC, bExecute := TRUE );
		step := 2;

	2:(* Wait until open not busy *)
		fbFileOpen( bExecute := FALSE, bError => bError, nErrID => nErrID, hFile => hFile );
		IF NOT fbFileOpen.bBusy THEN
			IF NOT fbFileOpen.bError THEN
				step := 3;
			ELSE(* Error: file not found? *)
				step := 100;
			END_IF
		END_IF
		
	3:(* Convert one PLC record to CSV format *)
		sCSVLine := '';
		fbWriter.eCmd := eEnumCmd_First;(* Write first field value *)
		
		FOR nColumn := 1 TO MAX_CSV_COLUMNS BY 1 DO
				
				IF nColumn = 1 THEN
					sCSVField := STRING_TO_CSVFIELD(sColumn1TimeStamp, FALSE);
				ELSIF nColumn = 2 THEN
					sCSVField := STRING_TO_CSVFIELD(sColumn2, FALSE);
				ELSIF nColumn = 3 THEN
					sCSVField := STRING_TO_CSVFIELD(sColumn3, FALSE);
				ELSIF nColumn = 4 THEN
					sCSVField := STRING_TO_CSVFIELD(sColumn4, FALSE);
				ELSIF nColumn = 5 THEN
					sCSVField := STRING_TO_CSVFIELD(sColumn5, FALSE);
				ELSIF nColumn = 6 THEN	
					sCSVField := STRING_TO_CSVFIELD(sColumn6, FALSE);
				ELSIF nColumn = 7 THEN	
					sCSVField := STRING_TO_CSVFIELD(sColumn7, FALSE);
				END_IF
				
				(* Add new field to the record buffer *)
				fbWriter( 	pBuffer := ADR( sCSVLine ), cbBuffer := SIZEOF( sCSVLine ) - 1, putValue := sCSVField, pValue := 0, cbValue := 0,
							bCRLF := ( nColumn = MAX_CSV_COLUMNS ) );
										
				IF fbWriter.bOk THEN
					fbWriter.eCmd := eEnumCmd_Next;(* Write next field value *)
				ELSE(* Error *)
					step := 100;
					RETURN;
				END_IF

		END_FOR

		(* FB_FilePuts adds allready CR (carriage return) to the written line.
		We have to replace the $R$L characters with $L character to avoid double CR. *)
		IF RIGHT( sCSVLine, 2 ) = '$R$L' THEN
			sCSVLine := REPLACE( sCSVLine, '$L', 2, LEN( sCSVLine ) - 1 );
		END_IF

		step := 4;(* Write record to the file *)
		
	4:	(* Write single text line *)
		fbFilePuts( bExecute := FALSE );
		fbFilePuts( sNetId := sNetId, hFile := hFile, sLine := sCSVLine, bExecute := TRUE );
		step := 5;

	5:(* Wait until write not busy *)
		fbFilePuts( bExecute := FALSE, bError => bError, nErrID => nErrID );
		IF NOT fbFilePuts.bBusy THEN
			IF NOT fbFilePuts.bError THEN
				step := 10;(* Close file *)
			ELSE(* Error *)
				step := 100;
			END_IF
		END_IF

	10:	(* Close source file *)
		fbFileClose( bExecute := FALSE );
		fbFileClose( sNetId := sNetId, hFile := hFile, bExecute := TRUE );
		step := 11;

	11:(* Wait until close not busy *)
		fbFileClose( bExecute := FALSE, bError => bError, nErrID => nErrID );
		IF ( NOT fbFileClose.bBusy ) THEN
			hFile := 0;
			step := 100;
		END_IF

	100: (* Error or ready step => cleanup *)
		IF ( hFile <> 0 ) THEN
			step := 10; (* Close the source file *)
		ELSE
			bBusy := FALSE;
			step := 0;	(* Ready *)
		END_IF

END_CASE

END_FUNCTION_BLOCK

// ---- POUs/Loggning/Temp_Logg.TcPOU
PROGRAM Temp_Logg
VAR
	
	fbLogg1 		:FB_SaveToCSV_Temp;
	tUpdateTime1	:TIME:=T#5S;
	sFileName1		:STRING(255):='Tempgivare';
	
	

END_VAR

fbLogg1(
	bChangeSeparatorToComma:= FALSE, 
	bExecute:= GVL_Fastighet.CSVTempProbes, 
	tUpdateTime:= tUpdateTime1, 
	sFileName:= sFileName1, 
	nDayOfWeek:= PLC_TID.fbTime.systemTime.wDayOfWeek,
	sColumn1TimeStamp:= PLC_TID.systemTime, 
	sColumn2:= REAL_TO_STRING(GVL_IO._GT41_MV), 
	sColumn3:= REAL_TO_STRING(GVL_IO._GT42_MV), 
	sColumn4:= REAL_TO_STRING(GVL_IO._GT43_MV), 
	sColumn5:= REAL_TO_STRING(GVL_IO._GT44_MV), 
	sColumn6:= REAL_TO_STRING(GVL_IO._GT45_MV), 
	sColumn7:= REAL_TO_STRING(GVL_IO._GT46_MV),
	sColumn8:= REAL_TO_STRING(GVL_IO._GT47_MV),
	sColumn9:= REAL_TO_STRING(GVL_IO._GT48_MV));

END_PROGRAM

// ---- POUs/_FBs/FB_SaveToCSV_Temp.TcPOU
FUNCTION_BLOCK FB_SaveToCSV_Temp
VAR CONSTANT
	MAX_CSV_COLUMNS 	: UDINT := 9;
END_VAR
VAR_INPUT
	(*	In USA/UK the CSV field separator is a comma.
	In Germany and some other European countries the CSV field separator is a semicolon. *)
	bChangeSeparatorToComma	: BOOL := FALSE;
	bExecute : BOOL;
	tUpdateTime : TIME:=T#1S; //Update time 
	sFileName	: T_MaxString := 'DefaultName';(* CSV destination file path and name *)
	nDayOfWeek : WORD;
	sColumn1TimeStamp : T_MaxString;
	sColumn2 : STRING;
	sColumn3 : STRING;
	sColumn4 : STRING; 
	sColumn5 : STRING;
	sColumn6 : STRING;
	sColumn7 : STRING;
	sColumn8 : STRING;
	sColumn9 : STRING;
END_VAR
VAR
	sNetId			: T_AmsNetId := '';	(* TwinCAT system network address *)	
	sCSVLine		: T_MaxString := '';(* Single CSV text line (row, record), we are using string as record buffer (your are able to see created fields) *)
	sCSVField		: T_MaxString := '';(* Single CSV field value (column, record field) *)
	bBusy			: BOOL;
	bError			: BOOL;
	nErrId			: UDINT;
	nColumn		: UDINT 	:= 1;(* Column number (record field) *)
	hFile			: UINT		:= 0;(* File handle of the source file *)
	step			: DWORD 	:= 0;
	fbFileOpen	: FB_FileOpen;(* Opens file *)
	fbFileClose	: FB_FileClose;(* Closes file *)
	fbFilePuts		: FB_FilePuts;(* Writes one record (line) *)
	fbWriter		: FB_CSVMemBufferWriter;(* Helper function block used to create CSV data bytes (single record line) *)	
	tUpdateTimer : TON;
	sCompleteFileName : STRING;
	sPathName : T_MaxString;
	sTempDate : STRING;
	sDate : STRING;
	bWeekUpdate : BOOL;
END_VAR

(* Call the timer every plc-cycle *)
tUpdateTimer(IN:=NOT tUpdateTimer.Q, PT:=tUpdateTime);


(* Update filename *)
IF nDayOfWeek = 1 AND bWeekUpdate THEN //1=Monday	
		sCompleteFileName	:= sFileName;
		sTempDate := DELETE(sColumn1TimeStamp, 16,11); //Cut the timestamp so we only save the date
		sDate := INSERT(sTempDate, '_', 10); //Add '-' after the date for seperation
		sPathName:=CONCAT(CONCAT('C:\Loggning\',CONCAT(sDate,sFileName)),'.csv');
		bWeekUpdate := FALSE;
ELSE
	(* Update if name has changed *)
	IF sCompleteFileName <> sFileName THEN
		sCompleteFileName := sFileName;
		sTempDate := DELETE(sColumn1TimeStamp, 16,11); //Cut the timestamp so we only save the date
		sDate := INSERT(sTempDate, '_', 10); //Add '-' after the date for seperation
		sPathName:=CONCAT(CONCAT('C:\Loggning\',CONCAT(sDate,sCompleteFileName)),'.csv');
	END_IF	
END_IF

IF nDayOfWeek <> 1 THEN
	bWeekUpdate := TRUE;
END_IF

CASE step OF
	0:	(* Wait for rising edge at bWrite variable *)
		IF bExecute AND tUpdateTimer.Q THEN
			bBusy 		:= TRUE;
			bError		:= FALSE;
			nErrId		:= 0;
			hFile			:= 0;
			step 		:= 1;
		END_IF

	1:	(* Open source file *)
		fbFileOpen(  bExecute := FALSE  );
		fbFileOpen( 	sNetId := sNetId, sPathName := sPathName, nMode := FOPEN_MODEAPPEND OR FOPEN_MODETEXT,(* Open file in TEXT mode! *)
						ePath := PATH_GENERIC, bExecute := TRUE );
		step := 2;

	2:(* Wait until open not busy *)
		fbFileOpen( bExecute := FALSE, bError => bError, nErrID => nErrID, hFile => hFile );
		IF NOT fbFileOpen.bBusy THEN
			IF NOT fbFileOpen.bError THEN
				step := 3;
			ELSE(* Error: file not found? *)
				step := 100;
			END_IF
		END_IF
		
	3:(* Convert one PLC record to CSV format *)
		sCSVLine := '';
		fbWriter.eCmd := eEnumCmd_First;(* Write first field value *)
		
		FOR nColumn := 1 TO MAX_CSV_COLUMNS BY 1 DO
				
				IF nColumn = 1 THEN
					sCSVField := STRING_TO_CSVFIELD(sColumn1TimeStamp, FALSE);
				ELSIF nColumn = 2 THEN
					sCSVField := STRING_TO_CSVFIELD(sColumn2, FALSE);
				ELSIF nColumn = 3 THEN
					sCSVField := STRING_TO_CSVFIELD(sColumn3, FALSE);
				ELSIF nColumn = 4 THEN
					sCSVField := STRING_TO_CSVFIELD(sColumn4, FALSE);
				ELSIF nColumn = 5 THEN
					sCSVField := STRING_TO_CSVFIELD(sColumn5, FALSE);
				ELSIF nColumn = 6 THEN	
					sCSVField := STRING_TO_CSVFIELD(sColumn6, FALSE);
				ELSIF nColumn = 7 THEN	
					sCSVField := STRING_TO_CSVFIELD(sColumn7, FALSE);
				ELSIF nColumn = 8 THEN	
					sCSVField := STRING_TO_CSVFIELD(sColumn8, FALSE);
				ELSIF nColumn = 9 THEN	
					sCSVField := STRING_TO_CSVFIELD(sColumn9, FALSE);
				END_IF
				
				(* Add new field to the record buffer *)
				fbWriter( 	pBuffer := ADR( sCSVLine ), cbBuffer := SIZEOF( sCSVLine ) - 1, putValue := sCSVField, pValue := 0, cbValue := 0,
							bCRLF := ( nColumn = MAX_CSV_COLUMNS ) );
										
				IF fbWriter.bOk THEN
					fbWriter.eCmd := eEnumCmd_Next;(* Write next field value *)
				ELSE(* Error *)
					step := 100;
					RETURN;
				END_IF

		END_FOR

		(* FB_FilePuts adds allready CR (carriage return) to the written line.
		We have to replace the $R$L characters with $L character to avoid double CR. *)
		IF RIGHT( sCSVLine, 2 ) = '$R$L' THEN
			sCSVLine := REPLACE( sCSVLine, '$L', 2, LEN( sCSVLine ) - 1 );
		END_IF

		step := 4;(* Write record to the file *)
		
	4:	(* Write single text line *)
		fbFilePuts( bExecute := FALSE );
		fbFilePuts( sNetId := sNetId, hFile := hFile, sLine := sCSVLine, bExecute := TRUE );
		step := 5;

	5:(* Wait until write not busy *)
		fbFilePuts( bExecute := FALSE, bError => bError, nErrID => nErrID );
		IF NOT fbFilePuts.bBusy THEN
			IF NOT fbFilePuts.bError THEN
				step := 10;(* Close file *)
			ELSE(* Error *)
				step := 100;
			END_IF
		END_IF

	10:	(* Close source file *)
		fbFileClose( bExecute := FALSE );
		fbFileClose( sNetId := sNetId, hFile := hFile, bExecute := TRUE );
		step := 11;

	11:(* Wait until close not busy *)
		fbFileClose( bExecute := FALSE, bError => bError, nErrID => nErrID );
		IF ( NOT fbFileClose.bBusy ) THEN
			hFile := 0;
			step := 100;
		END_IF

	100: (* Error or ready step => cleanup *)
		IF ( hFile <> 0 ) THEN
			step := 10; (* Close the source file *)
		ELSE
			bBusy := FALSE;
			step := 0;	(* Ready *)
		END_IF

END_CASE

END_FUNCTION_BLOCK

// ---- POUs/Loggning/SR05_Logg.TcPOU
PROGRAM SR05_Logg
VAR
	
	fbLogg1 		:FB_SaveToCSV_SR05;
	tUpdateTime1	:TIME:=T#5S;
	sFileName1		:STRING(255):='SR05Irr';
	
	

END_VAR

fbLogg1(
	bChangeSeparatorToComma:= FALSE, 
	bExecute:= GVL_Fastighet.CSVSR05, 
	tUpdateTime:= tUpdateTime1, 
	sFileName:= sFileName1, 
	nDayOfWeek:= PLC_TID.fbTime.systemTime.wDayOfWeek,
	sColumn1TimeStamp:= PLC_TID.systemTime, 
	sColumn2:= REAL_TO_STRING(GVL_SR05._SolarIrr), 
	sColumn3:= REAL_TO_STRING(GVL_SR05._BodyTemp), 
	sColumn4:= REAL_TO_STRING(GVL_SR05._ElecResistance), 
	sColumn5:= REAL_TO_STRING(GVL_SR05._VoltageOutput),);
	
	
	(*
 _SolarIrr				:REAL;			(*Solar Irradiance, signal in x 0.01 W/m², adr 2+3*)
_BodyTemp				:REAL;			(*Sensor body temperature in x 0.01 °C, adr 6*)
_ElecResistance			:REAL;			(*Sensor electrical resistance in x 0.1 Ω, adr 7*)	
_VoltageOutput			:REAL;			(*Solar Irradiance, signal in x 0.01 W/m², adr 2+3*)
*)

END_PROGRAM

// ---- POUs/_FBs/FB_SaveToCSV_SR05.TcPOU
FUNCTION_BLOCK FB_SaveToCSV_SR05
VAR CONSTANT
	MAX_CSV_COLUMNS 	: UDINT := 5;
END_VAR
VAR_INPUT
	(*	In USA/UK the CSV field separator is a comma.
	In Germany and some other European countries the CSV field separator is a semicolon. *)
	bChangeSeparatorToComma	: BOOL := FALSE;
	bExecute : BOOL;
	tUpdateTime : TIME:=T#5S; //Update time 
	sFileName	: T_MaxString := 'CSVSR05';(* CSV destination file path and name *)
	nDayOfWeek : WORD;
	sColumn1TimeStamp : T_MaxString;
	sColumn2 : STRING;
	sColumn3 : STRING;
	sColumn4 : STRING; 
	sColumn5 : STRING;
END_VAR
VAR
	sNetId			: T_AmsNetId := '';	(* TwinCAT system network address *)	
	sCSVLine		: T_MaxString := '';(* Single CSV text line (row, record), we are using string as record buffer (your are able to see created fields) *)
	sCSVField		: T_MaxString := '';(* Single CSV field value (column, record field) *)
	bBusy			: BOOL;
	bError			: BOOL;
	nErrId			: UDINT;
	nColumn		: UDINT 	:= 1;(* Column number (record field) *)
	hFile			: UINT		:= 0;(* File handle of the source file *)
	step			: DWORD 	:= 0;
	fbFileOpen	: FB_FileOpen;(* Opens file *)
	fbFileClose	: FB_FileClose;(* Closes file *)
	fbFilePuts		: FB_FilePuts;(* Writes one record (line) *)
	fbWriter		: FB_CSVMemBufferWriter;(* Helper function block used to create CSV data bytes (single record line) *)	
	tUpdateTimer : TON;
	sCompleteFileName : STRING;
	sPathName : T_MaxString;
	sTempDate : STRING;
	sDate : STRING;
	bWeekUpdate : BOOL;
END_VAR

(* Call the timer every plc-cycle *)
tUpdateTimer(IN:=NOT tUpdateTimer.Q, PT:=tUpdateTime);


(* Update filename *)
IF nDayOfWeek = 1 AND bWeekUpdate THEN //1=Monday	
		sCompleteFileName	:= sFileName;
		sTempDate := DELETE(sColumn1TimeStamp, 16,11); //Cut the timestamp so we only save the date
		sDate := INSERT(sTempDate, '_', 10); //Add '-' after the date for seperation
		sPathName:=CONCAT(CONCAT('C:\Loggning\SR05Irr\',CONCAT(sDate,sFileName)),'.csv');
		bWeekUpdate := FALSE;
ELSE
	(* Update if name has changed *)
	IF sCompleteFileName <> sFileName THEN
		sCompleteFileName := sFileName;
		sTempDate := DELETE(sColumn1TimeStamp, 16,11); //Cut the timestamp so we only save the date
		sDate := INSERT(sTempDate, '_', 10); //Add '-' after the date for seperation
		sPathName:=CONCAT(CONCAT('C:\Loggning\SR05Irr\',CONCAT(sDate,sCompleteFileName)),'.csv');
	END_IF	
END_IF

IF nDayOfWeek <> 1 THEN
	bWeekUpdate := TRUE;
END_IF

CASE step OF
	0:	(* Wait for rising edge at bWrite variable *)
		IF bExecute AND tUpdateTimer.Q THEN
			bBusy 		:= TRUE;
			bError		:= FALSE;
			nErrId		:= 0;
			hFile			:= 0;
			step 		:= 1;
		END_IF

	1:	(* Open source file *)
		fbFileOpen(  bExecute := FALSE  );
		fbFileOpen( 	sNetId := sNetId, sPathName := sPathName, nMode := FOPEN_MODEAPPEND OR FOPEN_MODETEXT,(* Open file in TEXT mode! *)
						ePath := PATH_GENERIC, bExecute := TRUE );
		step := 2;

	2:(* Wait until open not busy *)
		fbFileOpen( bExecute := FALSE, bError => bError, nErrID => nErrID, hFile => hFile );
		IF NOT fbFileOpen.bBusy THEN
			IF NOT fbFileOpen.bError THEN
				step := 3;
			ELSE(* Error: file not found? *)
				step := 100;
			END_IF
		END_IF
		
	3:(* Convert one PLC record to CSV format *)
		sCSVLine := '';
		fbWriter.eCmd := eEnumCmd_First;(* Write first field value *)
		
		FOR nColumn := 1 TO MAX_CSV_COLUMNS BY 1 DO
				
				IF nColumn = 1 THEN
					sCSVField := STRING_TO_CSVFIELD(sColumn1TimeStamp, FALSE);
				ELSIF nColumn = 2 THEN
					sCSVField := STRING_TO_CSVFIELD(sColumn2, FALSE);
				ELSIF nColumn = 3 THEN
					sCSVField := STRING_TO_CSVFIELD(sColumn3, FALSE);
				ELSIF nColumn = 4 THEN
					sCSVField := STRING_TO_CSVFIELD(sColumn4, FALSE);
				ELSIF nColumn = 5 THEN
					sCSVField := STRING_TO_CSVFIELD(sColumn5, FALSE);
				END_IF
				
				(* Add new field to the record buffer *)
				fbWriter( 	pBuffer := ADR( sCSVLine ), cbBuffer := SIZEOF( sCSVLine ) - 1, putValue := sCSVField, pValue := 0, cbValue := 0,
							bCRLF := ( nColumn = MAX_CSV_COLUMNS ) );
										
				IF fbWriter.bOk THEN
					fbWriter.eCmd := eEnumCmd_Next;(* Write next field value *)
				ELSE(* Error *)
					step := 100;
					RETURN;
				END_IF

		END_FOR

		(* FB_FilePuts adds allready CR (carriage return) to the written line.
		We have to replace the $R$L characters with $L character to avoid double CR. *)
		IF RIGHT( sCSVLine, 2 ) = '$R$L' THEN
			sCSVLine := REPLACE( sCSVLine, '$L', 2, LEN( sCSVLine ) - 1 );
		END_IF

		step := 4;(* Write record to the file *)
		
	4:	(* Write single text line *)
		fbFilePuts( bExecute := FALSE );
		fbFilePuts( sNetId := sNetId, hFile := hFile, sLine := sCSVLine, bExecute := TRUE );
		step := 5;

	5:(* Wait until write not busy *)
		fbFilePuts( bExecute := FALSE, bError => bError, nErrID => nErrID );
		IF NOT fbFilePuts.bBusy THEN
			IF NOT fbFilePuts.bError THEN
				step := 10;(* Close file *)
			ELSE(* Error *)
				step := 100;
			END_IF
		END_IF

	10:	(* Close source file *)
		fbFileClose( bExecute := FALSE );
		fbFileClose( sNetId := sNetId, hFile := hFile, bExecute := TRUE );
		step := 11;

	11:(* Wait until close not busy *)
		fbFileClose( bExecute := FALSE, bError => bError, nErrID => nErrID );
		IF ( NOT fbFileClose.bBusy ) THEN
			hFile := 0;
			step := 100;
		END_IF

	100: (* Error or ready step => cleanup *)
		IF ( hFile <> 0 ) THEN
			step := 10; (* Close the source file *)
		ELSE
			bBusy := FALSE;
			step := 0;	(* Ready *)
		END_IF

END_CASE

END_FUNCTION_BLOCK

// ---- POUs/Systemprogram/WatchDog_PLC.TcPOU
PROGRAM WatchDog_PLC
VAR
	TON_0: TON;
END_VAR

TON_0(IN := GVL_Larm._PLC_WD, PT := T#10s); // TON
GVL_Larm._PLC_WD := NOT (NOT TON_0.Q);

END_PROGRAM

// ---- POUs/Novram Hantering/NovramHandling.TcPOU
PROGRAM NovramHandling
VAR
	fbReadSaveNovram:FB_NovRamReadWrite;
	stData:ST_NovramData;
END_VAR

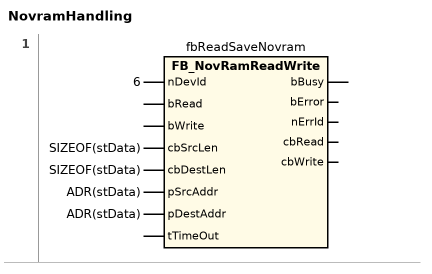
// NETWORK 1
fbReadSaveNovram(
    nDevId := 6,
    cbSrcLen := SIZEOF(stData),
    cbDestLen := SIZEOF(stData),
    pSrcAddr := ADR(stData),
    pDestAddr := ADR(stData)); // FB_NovRamReadWrite

END_PROGRAM

// ---- POUs/_FBs/FB_HUKSEFLUX_SR05.TcPOU

FUNCTION_BLOCK FB_HUKSEFLUX_SR05
VAR_INPUT
	bEnable:			BOOL;		(*Enable*)
	bySlaveAdr:			BYTE;		(*Slav Id*)
END_VAR
VAR_OUTPUT
	bBusy:					BOOL;		(*Upptagen med arbete*)
	bMbCommErr:				BOOL;		(*Modbus Komm. fel*)
	
	//_rIrr 					:REAL;			(*Solar Irradiance, signal in x 0.01 W/m², adr 2+3*)
	//_rBodyTemp				:REAL;			(*Sensor body temperature in x 0.01 °C, adr 6*)
	//_rElecResistance		:REAL;			(*Sensor electrical resistance in x 0.1 Ω, adr 7*)	
	//_rVoltageOutput			:REAL;			(*Solar Irradiance, signal in x 0.01 W/m², adr 2+3*)
	
	
END_VAR
VAR
	fbRtuMaster:		ModbusRtuMaster_KL6x22B; 		(*Modbus master instans*)
	fbDelay:			TON;							(*Fördröjning mellan sekvenserna*)
	nStat:				INT := 0;						(*Sekvens*)
	
stSR05_Data:ST_SR05_IrrMeter;	
	
END_VAR

CASE nStat OF

0:(*Start steg*)
	IF bEnable THEN
		bMbCommErr := FALSE;
		bBusy := TRUE;
		nStat := 2;
	END_IF


2:(*Modbus Funktion 3, Läs data från Holding Registers*)
fbRtuMaster.ReadRegs(
					UnitID:= bySlaveAdr ,
					Quantity:= 2,
					MBAddr:= 2 ,
					cbLength:= SIZEOF(stSR05_Data.Solar_Irradiance_raw) , // Solar irradiance value from sensor, needs to be recalculated to W/m2 acc to formula in manual
					pMemoryAddr:=  ADR(stSR05_Data.Solar_Irradiance_raw),
					Execute:= TRUE ,
					Timeout:= T#2S ,BUSY=> ,	Error=> , ErrorId=> ,cbRead=> );
					
					
IF fbRtuMaster.Error THEN
	nStat := 999;
ELSIF  NOT fbRtuMaster.BUSY AND NOT fbRtuMaster.Error THEN
	fbRtuMaster.ReadRegs(Execute := FALSE);
	nStat := 3;
END_IF


3:	(*Fördröj*)
fbDelay(IN:= TRUE, PT:=T#100ms , Q=> , ET=> );
IF fbDelay.Q THEN
	fbDelay(IN:= FALSE);
	nStat := 4;
END_IF;


4:(*Modbus Funktion 3, Läs data från Holding Registers*)
fbRtuMaster.ReadRegs(
					UnitID:= bySlaveAdr ,
					Quantity:= 1,
					MBAddr:= 6 ,
					cbLength:= SIZEOF(stSR05_Data.Sensor_Body_Temp) ,
					pMemoryAddr:=  ADR(stSR05_Data.Sensor_Body_Temp),
					Execute:= TRUE ,
					Timeout:= T#2s ,BUSY=> ,	Error=> , ErrorId=> ,cbRead=> );

IF fbRtuMaster.Error THEN
	nStat := 999;
ELSIF  NOT fbRtuMaster.BUSY AND NOT fbRtuMaster.Error THEN
	fbRtuMaster.ReadRegs(Execute := FALSE);
	nStat := 5;
END_IF


5:	(*Fördröj*)
fbDelay(IN:= TRUE, PT:=T#100ms , Q=> , ET=> );
IF fbDelay.Q THEN
	fbDelay(IN:= FALSE);
	nStat := 6;
END_IF;


4:(*Modbus Funktion 3, Läs data från Holding Registers*)
fbRtuMaster.ReadRegs(
					UnitID:= bySlaveAdr ,
					Quantity:= 1,
					MBAddr:= 7 ,
					cbLength:= SIZEOF(stSR05_Data.Sensor_Elec_Resistance) ,
					pMemoryAddr:=  ADR(stSR05_Data.Sensor_Elec_Resistance),
					Execute:= TRUE ,
					Timeout:= T#2s ,BUSY=> ,	Error=> , ErrorId=> ,cbRead=> );

IF fbRtuMaster.Error THEN
	nStat := 999;
ELSIF  NOT fbRtuMaster.BUSY AND NOT fbRtuMaster.Error THEN
	fbRtuMaster.ReadRegs(Execute := FALSE);
	nStat := 7;
END_IF


7:	(*Fördröj*)
fbDelay(IN:= TRUE, PT:=T#100ms , Q=> , ET=> );
IF fbDelay.Q THEN
	fbDelay(IN:= FALSE);
	nStat := 8;
END_IF;


2:(*Modbus Funktion 3, Läs data från Holding Registers*)
fbRtuMaster.ReadRegs(
					UnitID:= bySlaveAdr ,
					Quantity:= 2,
					MBAddr:= 10 ,
					cbLength:= SIZEOF(stSR05_Data.Sensor_voltage_output) ,
					pMemoryAddr:=  ADR(stSR05_Data.Sensor_voltage_output),
					Execute:= TRUE ,
					Timeout:= T#2s ,BUSY=> ,	Error=> , ErrorId=> ,cbRead=> );

IF fbRtuMaster.Error THEN
	nStat := 999;
ELSIF  NOT fbRtuMaster.BUSY AND NOT fbRtuMaster.Error THEN
	fbRtuMaster.ReadRegs(Execute := FALSE);
	nStat := 20;
END_IF



20:(*Läsning klar*)
	(*Beräkna och visa på utgången*)
	
	//Calculation of Solar irradiance acc to SR05 Manual v1610, see page 43 
	stSR05_Data.Solar_Irradiance:= ((DWORD TO WORD (stSR05_Data.Solar_Irradiance_raw)* (2 EXP 16) )+ DWORD_TO_WORD( SHR(stSR05_Data.Solar_Irradiance_raw, 16 )));  
	
	//
	GVL_SR05._SolarIrr:=		stSR05_Data.Solar_Irradiance * 0.01; //Signal in x 0.01 W/m², scaled here to W/m²
	GVL_SR05._BodyTemp:=		stSR05_Data.Sensor_Body_Temp * 0.01; //Signal in x 0.01 °C, scaled here to Celsius (°C)
	GVL_SR05._ElecResistance:=	stSR05_Data.Sensor_Elec_Resistance * 0.1; //Signal in x 0.1 Ω, scaled here to Ω
	GVL_SR05._VoltageOutput:=	stSR05_Data.Sensor_voltage_output * 10* EXP(-9); //Signal in x 10-9 V, scaled here to V
	
	(*Scale and store in Global variables*)
	//GVL_SR05._Irr:= 
	
	nStat := 0;

999:(*Något blev fel*)
	fbRtuMaster.ReadRegs(Execute := FALSE);
	bMbCommErr:= TRUE;
	bBusy := FALSE;
	nStat := 0;
END_CASE

END_FUNCTION_BLOCK
